LIN {X 0,Y 247.82,Z 1220.634,A -85,B 0,C 180,E1 25956.529,E2 25956.529} C_VEL
LIN {X 0,Y 211.534,Z 1249.474,A -85,B 0,C 180,E1 25974.763,E2 25974.763} C_VEL
LIN {X 0,Y 196.821,Z 1262.562,A -85,B 0,C 180,E1 25994.337,E2 25994.337} C_VEL
LIN {X 0,Y 195.288,Z 1265.442,A -85,B 0,C 180,E1 26012.226,E2 26012.226} C_VEL
LIN {X 0,Y 199.92,Z 1259.369,A -85,B 0,C 180,E1 26032.313,E2 26032.313} C_VEL
LIN {X 0,Y 222.937,Z 1240.033,A -85,B 0,C 180,E1 26052.917,E2 26052.917} C_VEL
LIN {X 0,Y 264.688,Z 1206.28,A -85,B 0,C 180,E1 26068.603,E2 26068.603} C_VEL
LIN {X 0,Y 314.502,Z 1158.82,A -85,B 0,C 180,E1 26078.95,E2 26078.95} C_VEL
LIN {X 0,Y 361.028,Z 1101.859,A -85,B 0,C 180,E1 26085.304,E2 26085.304} C_VEL
LIN {X 0,Y 364.505,Z 1096.146,A -85,B 0,C 180,E1 26086.175,E2 26086.175} C_VEL
LIN {X 0,Y 366.989,Z 1082.941,A -85,B 0,C 180,E1 26094.136,E2 26094.136} C_VEL
LIN {X 0,Y 368.189,Z 1080.031,A -85,B 0,C 180,E1 26101.248,E2 26101.248} C_VEL
LIN {X 0,Y 367.729,Z 1090.519,A -85,B 0,C 180,E1 26110.168,E2 26110.168} C_VEL
LIN {X 0,Y 366.404,Z 1098.087,A -85,B 0,C 180,E1 26113.18,E2 26113.18} C_VEL
LIN {X 0,Y 318.911,Z 1159.271,A -85,B 0,C 180,E1 26119.202,E2 26119.202} C_VEL
LIN {X 0,Y 268.992,Z 1209.566,A -85,B 0,C 180,E1 26128.983,E2 26128.983} C_VEL
LIN {X 0,Y 226.358,Z 1246.346,A -85,B 0,C 180,E1 26143.867,E2 26143.867} C_VEL
LIN {X 0,Y 201.739,Z 1268.464,A -85,B 0,C 180,E1 26163.161,E2 26163.161} C_VEL
LIN {X 0,Y 195.076,Z 1277.751,A -85,B 0,C 180,E1 26183.298,E2 26183.298} C_VEL
LIN {X 0,Y 195.027,Z 1277.758,A -85,B 0,C 180,E1 26196.707,E2 26196.707} C_VEL
LIN {X 0,Y 200.195,Z 1270.124,A -85,B 0,C 180,E1 26214.652,E2 26214.652} C_VEL
LIN {X 0,Y 224.432,Z 1247.98,A -85,B 0,C 180,E1 26235.257,E2 26235.257} C_VEL
LIN {X 0,Y 267.615,Z 1210.892,A -85,B 0,C 180,E1 26250.716,E2 26250.716} C_VEL
LIN {X 0,Y 318.076,Z 1160.468,A -85,B 0,C 180,E1 26260.642,E2 26260.642} C_VEL
LIN {X 0,Y 365.292,Z 1100.027,A -85,B 0,C 180,E1 26266.725,E2 26266.725} C_VEL
LIN {X 0,Y 367.584,Z 1095.292,A -85,B 0,C 180,E1 26267.566,E2 26267.566} C_VEL
LIN {X 0,Y 368.085,Z 1083.099,A -85,B 0,C 180,E1 26275.203,E2 26275.203} C_VEL
LIN {X 0,Y 368.206,Z 1079.906,A -85,B 0,C 180,E1 26281.113,E2 26281.113} C_VEL
LIN {X 0,Y 365.81,Z 1089.05,A -85,B 0,C 180,E1 26290.07,E2 26290.07} C_VEL
LIN {X 0,Y 364.059,Z 1097.903,A -85,B 0,C 180,E1 26294.235,E2 26294.235} C_VEL
LIN {X 0,Y 316.416,Z 1157.039,A -85,B 0,C 180,E1 26300.676,E2 26300.676} C_VEL
LIN {X 0,Y 267.993,Z 1203.645,A -85,B 0,C 180,E1 26310.453,E2 26310.453} C_VEL
LIN {X 0,Y 247.82,Z 1220.634,A -85,B 0,C 180,E1 26316.529,E2 26316.529} C_VEL
LIN {X 0,Y 224.197,Z 1234.966,A -85,B 0,C 180,E1 26321.962,E2 26321.962} C_VEL
LIN {X 0,Y 195.817,Z 1256.691,A -85,B 0,C 180,E1 26341.874,E2 26341.874} C_VEL
LIN {X 0,Y 187.278,Z 1265.309,A -85,B 0,C 180,E1 26363.015,E2 26363.015} C_VEL
LIN {X 0,Y 187.314,Z 1265.279,A -85,B 0,C 180,E1 26376.981,E2 26376.981} C_VEL
LIN {X 0,Y 195.871,Z 1256.598,A -85,B 0,C 180,E1 26398.128,E2 26398.128} C_VEL
LIN {X 0,Y 226.431,Z 1233.395,A -85,B 0,C 180,E1 26418.751,E2 26418.751} C_VEL
LIN {X 0,Y 272.513,Z 1196.349,A -85,B 0,C 180,E1 26433.039,E2 26433.039} C_VEL
LIN {X 0,Y 322.853,Z 1146.97,A -85,B 0,C 180,E1 26442.044,E2 26442.044} C_VEL
LIN {X 0,Y 359.4,Z 1101.578,A -85,B 0,C 180,E1 26446.646,E2 26446.646} C_VEL
LIN {X 0,Y 362.111,Z 1089.495,A -85,B 0,C 180,E1 26454.057,E2 26454.057} C_VEL
LIN {X 0,Y 363.545,Z 1086.616,A -85,B 0,C 180,E1 26461.264,E2 26461.264} C_VEL
LIN {X 0,Y 362.693,Z 1097.481,A -85,B 0,C 180,E1 26470.384,E2 26470.384} C_VEL
LIN {X 0,Y 361.222,Z 1102.92,A -85,B 0,C 180,E1 26472.285,E2 26472.285} C_VEL
LIN {X 0,Y 311.998,Z 1163.707,A -85,B 0,C 180,E1 26478.411,E2 26478.411} C_VEL
LIN {X 0,Y 260.983,Z 1212.827,A -85,B 0,C 180,E1 26488.383,E2 26488.383} C_VEL
LIN {X 0,Y 216.361,Z 1249.506,A -85,B 0,C 180,E1 26504.481,E2 26504.481} C_VEL
LIN {X 0,Y 191.903,Z 1270.717,A -85,B 0,C 180,E1 26525.708,E2 26525.708} C_VEL
LIN {X 0,Y 187.07,Z 1277.486,A -85,B 0,C 180,E1 26543.01,E2 26543.01} C_VEL
LIN {X 0,Y 187.026,Z 1277.494,A -85,B 0,C 180,E1 26556.995,E2 26556.995} C_VEL
LIN {X 0,Y 192.685,Z 1269.852,A -85,B 0,C 180,E1 26575.681,E2 26575.681} C_VEL
LIN {X 0,Y 218.587,Z 1247.704,A -85,B 0,C 180,E1 26596.824,E2 26596.824} C_VEL
LIN {X 0,Y 263.616,Z 1210.619,A -85,B 0,C 180,E1 26612.305,E2 26612.305} C_VEL
LIN {X 0,Y 315.195,Z 1160.441,A -85,B 0,C 180,E1 26622.038,E2 26622.038} C_VEL
LIN {X 0,Y 362.594,Z 1100.59,A -85,B 0,C 180,E1 26628.16,E2 26628.16} C_VEL
LIN {X 0,Y 363.313,Z 1088.664,A -85,B 0,C 180,E1 26636.34,E2 26636.34} C_VEL
LIN {X 0,Y 363.54,Z 1086.485,A -85,B 0,C 180,E1 26641.127,E2 26641.127} C_VEL
LIN {X 0,Y 360.795,Z 1095.869,A -85,B 0,C 180,E1 26650.224,E2 26650.224} C_VEL
LIN {X 0,Y 358.316,Z 1103.36,A -85,B 0,C 180,E1 26653.395,E2 26653.395} C_VEL
LIN {X 0,Y 310.157,Z 1160.831,A -85,B 0,C 180,E1 26659.809,E2 26659.809} C_VEL
LIN {X 0,Y 259.129,Z 1207.77,A -85,B 0,C 180,E1 26670.113,E2 26670.113} C_VEL
LIN {X 0,Y 224.197,Z 1234.966,A -85,B 0,C 180,E1 26681.962,E2 26681.962} C_VEL
LIN {X 0,Y 202.634,Z 1246.721,A -85,B 0,C 180,E1 26688.863,E2 26688.863} C_VEL
LIN {X 0,Y 183.451,Z 1261.13,A -85,B 0,C 180,E1 26708.135,E2 26708.135} C_VEL
LIN {X 0,Y 179.089,Z 1265.984,A -85,B 0,C 180,E1 26727.569,E2 26727.569} C_VEL
LIN {X 0,Y 181.319,Z 1263.044,A -85,B 0,C 180,E1 26747.039,E2 26747.039} C_VEL
LIN {X 0,Y 200.823,Z 1247.851,A -85,B 0,C 180,E1 26769.981,E2 26769.981} C_VEL
LIN {X 0,Y 242.467,Z 1217.738,A -85,B 0,C 180,E1 26787.99,E2 26787.99} C_VEL
LIN {X 0,Y 294.507,Z 1173.617,A -85,B 0,C 180,E1 26799.507,E2 26799.507} C_VEL
LIN {X 0,Y 345.516,Z 1117.781,A -85,B 0,C 180,E1 26806.587,E2 26806.587} C_VEL
LIN {X 0,Y 354.577,Z 1105.763,A -85,B 0,C 180,E1 26807.709,E2 26807.709} C_VEL
LIN {X 0,Y 357.614,Z 1094.475,A -85,B 0,C 180,E1 26816.024,E2 26816.024} C_VEL
LIN {X 0,Y 358.71,Z 1093.075,A -85,B 0,C 180,E1 26821.281,E2 26821.281} C_VEL
LIN {X 0,Y 357.6,Z 1104.102,A -85,B 0,C 180,E1 26830.46,E2 26830.46} C_VEL
LIN {X 0,Y 354.697,Z 1109.234,A -85,B 0,C 180,E1 26831.485,E2 26831.485} C_VEL
LIN {X 0,Y 304.591,Z 1168.393,A -85,B 0,C 180,E1 26837.656,E2 26837.656} C_VEL
LIN {X 0,Y 252.665,Z 1216.169,A -85,B 0,C 180,E1 26847.835,E2 26847.835} C_VEL
LIN {X 0,Y 207.148,Z 1251.806,A -85,B 0,C 180,E1 26864.675,E2 26864.675} C_VEL
LIN {X 0,Y 184.346,Z 1270.499,A -85,B 0,C 180,E1 26884.752,E2 26884.752} C_VEL
LIN {X 0,Y 179.063,Z 1277.221,A -85,B 0,C 180,E1 26902.695,E2 26902.695} C_VEL
LIN {X 0,Y 179.022,Z 1277.229,A -85,B 0,C 180,E1 26917.309,E2 26917.309} C_VEL
LIN {X 0,Y 185.224,Z 1269.58,A -85,B 0,C 180,E1 26936.796,E2 26936.796} C_VEL
LIN {X 0,Y 212.914,Z 1247.429,A -85,B 0,C 180,E1 26958.477,E2 26958.477} C_VEL
LIN {X 0,Y 259.603,Z 1210.534,A -85,B 0,C 180,E1 26973.896,E2 26973.896} C_VEL
LIN {X 0,Y 312.717,Z 1160.17,A -85,B 0,C 180,E1 26983.496,E2 26983.496} C_VEL
LIN {X 0,Y 357.527,Z 1105.477,A -85,B 0,C 180,E1 26988.92,E2 26988.92} C_VEL
LIN {X 0,Y 358.49,Z 1095.118,A -85,B 0,C 180,E1 26996.29,E2 26996.29} C_VEL
LIN {X 0,Y 358.707,Z 1092.939,A -85,B 0,C 180,E1 27001.142,E2 27001.142} C_VEL
LIN {X 0,Y 355.546,Z 1102.56,A -85,B 0,C 180,E1 27010.377,E2 27010.377} C_VEL
LIN {X 0,Y 354.073,Z 1106.906,A -85,B 0,C 180,E1 27012.377,E2 27012.377} C_VEL
LIN {X 0,Y 304.521,Z 1164.053,A -85,B 0,C 180,E1 27018.809,E2 27018.809} C_VEL
LIN {X 0,Y 252.236,Z 1210.301,A -85,B 0,C 180,E1 27029.224,E2 27029.224} C_VEL
LIN {X 0,Y 207.365,Z 1243.323,A -85,B 0,C 180,E1 27045.932,E2 27045.932} C_VEL
LIN {X 0,Y 202.634,Z 1246.721,A -85,B 0,C 180,E1 27048.863,E2 27048.863} C_VEL
LIN {X 0,Y 183.392,Z 1255.903,A -85,B 0,C 180,E1 27057.335,E2 27057.335} C_VEL
LIN {X 0,Y 171.965,Z 1264.872,A -85,B 0,C 180,E1 27077.248,E2 27077.248} C_VEL
LIN {X 0,Y 171.252,Z 1266.232,A -85,B 0,C 180,E1 27092.539,E2 27092.539} C_VEL
LIN {X 0,Y 177.324,Z 1260.268,A -85,B 0,C 180,E1 27115.128,E2 27115.128} C_VEL
LIN {X 0,Y 205.419,Z 1240.853,A -85,B 0,C 180,E1 27137.647,E2 27137.647} C_VEL
LIN {X 0,Y 253.016,Z 1206.793,A -85,B 0,C 180,E1 27153.526,E2 27153.526} C_VEL
LIN {X 0,Y 307.106,Z 1159.027,A -85,B 0,C 180,E1 27163.364,E2 27163.364} C_VEL
LIN {X 0,Y 349.8,Z 1110.023,A -85,B 0,C 180,E1 27168.818,E2 27168.818} C_VEL
LIN {X 0,Y 352.834,Z 1100.625,A -85,B 0,C 180,E1 27176.373,E2 27176.373} C_VEL
LIN {X 0,Y 353.886,Z 1099.52,A -85,B 0,C 180,E1 27181.299,E2 27181.299} C_VEL
LIN {X 0,Y 352.404,Z 1109.662,A -85,B 0,C 180,E1 27190.053,E2 27190.053} C_VEL
LIN {X 0,Y 300.349,Z 1169.933,A -85,B 0,C 180,E1 27196.404,E2 27196.404} C_VEL
LIN {X 0,Y 246.438,Z 1217.829,A -85,B 0,C 180,E1 27206.72,E2 27206.72} C_VEL
LIN {X 0,Y 199.799,Z 1252.653,A -85,B 0,C 180,E1 27223.796,E2 27223.796} C_VEL
LIN {X 0,Y 174.925,Z 1271.959,A -85,B 0,C 180,E1 27247.013,E2 27247.013} C_VEL
LIN {X 0,Y 171.215,Z 1277.464,A -85,B 0,C 180,E1 27267.461,E2 27267.461} C_VEL
LIN {X 0,Y 171.634,Z 1275.862,A -85,B 0,C 180,E1 27282.777,E2 27282.777} C_VEL
LIN {X 0,Y 184.77,Z 1263.609,A -85,B 0,C 180,E1 27305.855,E2 27305.855} C_VEL
LIN {X 0,Y 223.269,Z 1235.666,A -85,B 0,C 180,E1 27326.404,E2 27326.404} C_VEL
LIN {X 0,Y 275.503,Z 1193.538,A -85,B 0,C 180,E1 27339.512,E2 27339.512} C_VEL
LIN {X 0,Y 328.814,Z 1139.598,A -85,B 0,C 180,E1 27347.25,E2 27347.25} C_VEL
LIN {X 0,Y 352.52,Z 1109.78,A -85,B 0,C 180,E1 27349.969,E2 27349.969} C_VEL
LIN {X 0,Y 353.968,Z 1099.785,A -85,B 0,C 180,E1 27358.701,E2 27358.701} C_VEL
LIN {X 0,Y 352.024,Z 1103.065,A -85,B 0,C 180,E1 27366.114,E2 27366.114} C_VEL
LIN {X 0,Y 348.563,Z 1112.301,A -85,B 0,C 180,E1 27371.487,E2 27371.487} C_VEL
LIN {X 0,Y 296.977,Z 1169.258,A -85,B 0,C 180,E1 27378.071,E2 27378.071} C_VEL
LIN {X 0,Y 244.238,Z 1213.752,A -85,B 0,C 180,E1 27388.599,E2 27388.599} C_VEL
LIN {X 0,Y 198.822,Z 1245.441,A -85,B 0,C 180,E1 27405.798,E2 27405.798} C_VEL
LIN {X 0,Y 183.392,Z 1255.903,A -85,B 0,C 180,E1 27417.335,E2 27417.335} C_VEL
LIN {X 0,Y 167.503,Z 1262.23,A -85,B 0,C 180,E1 27427.557,E2 27427.557} C_VEL
LIN {X 0,Y 163.087,Z 1266.509,A -85,B 0,C 180,E1 27447.331,E2 27447.331} C_VEL
LIN {X 0,Y 164.522,Z 1264.699,A -85,B 0,C 180,E1 27465.063,E2 27465.063} C_VEL
LIN {X 0,Y 182.018,Z 1252.531,A -85,B 0,C 180,E1 27488.72,E2 27488.72} C_VEL
LIN {X 0,Y 223.224,Z 1225.893,A -85,B 0,C 180,E1 27508.221,E2 27508.221} C_VEL
LIN {X 0,Y 275.947,Z 1185.814,A -85,B 0,C 180,E1 27520.409,E2 27520.409} C_VEL
LIN {X 0,Y 329.244,Z 1133.47,A -85,B 0,C 180,E1 27527.862,E2 27527.862} C_VEL
LIN {X 0,Y 345.057,Z 1114.374,A -85,B 0,C 180,E1 27529.945,E2 27529.945} C_VEL
LIN {X 0,Y 348.705,Z 1105.384,A -85,B 0,C 180,E1 27538.845,E2 27538.845} C_VEL
LIN {X 0,Y 347.695,Z 1111.993,A -85,B 0,C 180,E1 27547.587,E2 27547.587} C_VEL
LIN {X 0,Y 346.201,Z 1116.091,A -85,B 0,C 180,E1 27549.381,E2 27549.381} C_VEL
LIN {X 0,Y 293.651,Z 1174.078,A -85,B 0,C 180,E1 27555.5,E2 27555.5} C_VEL
LIN {X 0,Y 239.428,Z 1220.197,A -85,B 0,C 180,E1 27565.775,E2 27565.775} C_VEL
LIN {X 0,Y 192.133,Z 1253.758,A -85,B 0,C 180,E1 27583.042,E2 27583.042} C_VEL
LIN {X 0,Y 167.404,Z 1271.689,A -85,B 0,C 180,E1 27605.917,E2 27605.917} C_VEL
LIN {X 0,Y 163.19,Z 1277.2,A -85,B 0,C 180,E1 27627.336,E2 27627.336} C_VEL
LIN {X 0,Y 163.731,Z 1275.596,A -85,B 0,C 180,E1 27643.405,E2 27643.405} C_VEL
LIN {X 0,Y 178.813,Z 1262.852,A -85,B 0,C 180,E1 27667.992,E2 27667.992} C_VEL
LIN {X 0,Y 220.389,Z 1234.213,A -85,B 0,C 180,E1 27688.783,E2 27688.783} C_VEL
LIN {X 0,Y 274.235,Z 1191.905,A -85,B 0,C 180,E1 27701.446,E2 27701.446} C_VEL
LIN {X 0,Y 328.798,Z 1137.381,A -85,B 0,C 180,E1 27708.862,E2 27708.862} C_VEL
LIN {X 0,Y 347.578,Z 1114.028,A -85,B 0,C 180,E1 27711.139,E2 27711.139} C_VEL
LIN {X 0,Y 348.89,Z 1106.026,A -85,B 0,C 180,E1 27718.683,E2 27718.683} C_VEL
LIN {X 0,Y 346.809,Z 1109.446,A -85,B 0,C 180,E1 27726.206,E2 27726.206} C_VEL
LIN {X 0,Y 343.981,Z 1116.331,A -85,B 0,C 180,E1 27730.466,E2 27730.466} C_VEL
LIN {X 0,Y 291.649,Z 1172.1,A -85,B 0,C 180,E1 27736.964,E2 27736.964} C_VEL
LIN {X 0,Y 238.969,Z 1214.983,A -85,B 0,C 180,E1 27747.201,E2 27747.201} C_VEL
LIN {X 0,Y 193.421,Z 1245.414,A -85,B 0,C 180,E1 27763.783,E2 27763.783} C_VEL
LIN {X 0,Y 167.503,Z 1262.23,A -85,B 0,C 180,E1 27787.557,E2 27787.557} C_VEL
LIN {X 0,Y 155.495,Z 1265.989,A -85,B 0,C 180,E1 27799.357,E2 27799.357} C_VEL
LIN {X 0,Y 155.363,Z 1266.338,A -85,B 0,C 180,E1 27818.427,E2 27818.427} C_VEL
LIN {X 0,Y 167.147,Z 1257.93,A -85,B 0,C 180,E1 27843.019,E2 27843.019} C_VEL
LIN {X 0,Y 206.316,Z 1234.282,A -85,B 0,C 180,E1 27865.871,E2 27865.871} C_VEL
LIN {X 0,Y 260.188,Z 1196.663,A -85,B 0,C 180,E1 27879.779,E2 27879.779} C_VEL
LIN {X 0,Y 315.943,Z 1146.366,A -85,B 0,C 180,E1 27887.952,E2 27887.952} C_VEL
LIN {X 0,Y 339.961,Z 1119.245,A -85,B 0,C 180,E1 27890.746,E2 27890.746} C_VEL
LIN {X 0,Y 343.594,Z 1111.606,A -85,B 0,C 180,E1 27898.832,E2 27898.832} C_VEL
LIN {X 0,Y 342.731,Z 1116.701,A -85,B 0,C 180,E1 27906.427,E2 27906.427} C_VEL
LIN {X 0,Y 340.761,Z 1120.982,A -85,B 0,C 180,E1 27908.405,E2 27908.405} C_VEL
LIN {X 0,Y 286.348,Z 1178.518,A -85,B 0,C 180,E1 27914.64,E2 27914.64} C_VEL
LIN {X 0,Y 231.031,Z 1223.386,A -85,B 0,C 180,E1 27925.127,E2 27925.127} C_VEL
LIN {X 0,Y 182.577,Z 1255.896,A -85,B 0,C 180,E1 27943.32,E2 27943.32} C_VEL
LIN {X 0,Y 158.534,Z 1272.684,A -85,B 0,C 180,E1 27967.48,E2 27967.48} C_VEL
LIN {X 0,Y 155.186,Z 1276.937,A -85,B 0,C 180,E1 27987.198,E2 27987.198} C_VEL
LIN {X 0,Y 155.82,Z 1275.329,A -85,B 0,C 180,E1 28004.099,E2 28004.099} C_VEL
LIN {X 0,Y 172.329,Z 1262.579,A -85,B 0,C 180,E1 28029.696,E2 28029.696} C_VEL
LIN {X 0,Y 215.441,Z 1234.41,A -85,B 0,C 180,E1 28050.479,E2 28050.479} C_VEL
LIN {X 0,Y 271.676,Z 1191.631,A -85,B 0,C 180,E1 28063.128,E2 28063.128} C_VEL
LIN {X 0,Y 327.296,Z 1137.112,A -85,B 0,C 180,E1 28070.287,E2 28070.287} C_VEL
LIN {X 0,Y 342.517,Z 1118.724,A -85,B 0,C 180,E1 28072.134,E2 28072.134} C_VEL
LIN {X 0,Y 343.762,Z 1112.266,A -85,B 0,C 180,E1 28078.663,E2 28078.663} C_VEL
LIN {X 0,Y 342.129,Z 1114.45,A -85,B 0,C 180,E1 28084.888,E2 28084.888} C_VEL
LIN {X 0,Y 339.03,Z 1120.817,A -85,B 0,C 180,E1 28089.466,E2 28089.466} C_VEL
LIN {X 0,Y 284.444,Z 1176.685,A -85,B 0,C 180,E1 28096.116,E2 28096.116} C_VEL
LIN {X 0,Y 229.669,Z 1219.072,A -85,B 0,C 180,E1 28106.827,E2 28106.827} C_VEL
LIN {X 0,Y 182.459,Z 1248.784,A -85,B 0,C 180,E1 28124.988,E2 28124.988} C_VEL
LIN {X 0,Y 158.066,Z 1263.894,A -85,B 0,C 180,E1 28150.356,E2 28150.356} C_VEL
LIN {X 0,Y 155.495,Z 1265.989,A -85,B 0,C 180,E1 28159.357,E2 28159.357} C_VEL
LIN {X 0,Y 147.144,Z 1267.023,A -85,B 0,C 180,E1 28172.526,E2 28172.526} C_VEL
LIN {X 0,Y 153.59,Z 1262.14,A -85,B 0,C 180,E1 28196.408,E2 28196.408} C_VEL
LIN {X 0,Y 185,Z 1244.276,A -85,B 0,C 180,E1 28221.219,E2 28221.219} C_VEL
LIN {X 0,Y 236.27,Z 1212.304,A -85,B 0,C 180,E1 28237.409,E2 28237.409} C_VEL
LIN {X 0,Y 294.045,Z 1166.277,A -85,B 0,C 180,E1 28247.02,E2 28247.02} C_VEL
LIN {X 0,Y 335.073,Z 1123.776,A -85,B 0,C 180,E1 28251.822,E2 28251.822} C_VEL
LIN {X 0,Y 338.374,Z 1117.761,A -85,B 0,C 180,E1 28258.819,E2 28258.819} C_VEL
LIN {X 0,Y 337.028,Z 1123.748,A -85,B 0,C 180,E1 28267.186,E2 28267.186} C_VEL
LIN {X 0,Y 280.986,Z 1181.213,A -85,B 0,C 180,E1 28273.47,E2 28273.47} C_VEL
LIN {X 0,Y 222.866,Z 1226.333,A -85,B 0,C 180,E1 28284.348,E2 28284.348} C_VEL
LIN {X 0,Y 174.905,Z 1256.809,A -85,B 0,C 180,E1 28302.46,E2 28302.46} C_VEL
LIN {X 0,Y 149.72,Z 1273.343,A -85,B 0,C 180,E1 28329.215,E2 28329.215} C_VEL
LIN {X 0,Y 147.157,Z 1276.673,A -85,B 0,C 180,E1 28347.045,E2 28347.045} C_VEL
LIN {X 0,Y 147.952,Z 1275.062,A -85,B 0,C 180,E1 28364.866,E2 28364.866} C_VEL
LIN {X 0,Y 165.982,Z 1262.306,A -85,B 0,C 180,E1 28391.539,E2 28391.539} C_VEL
LIN {X 0,Y 210.575,Z 1234.685,A -85,B 0,C 180,E1 28412.22,E2 28412.22} C_VEL
LIN {X 0,Y 267.272,Z 1193.074,A -85,B 0,C 180,E1 28424.517,E2 28424.517} C_VEL
LIN {X 0,Y 323.749,Z 1139.311,A -85,B 0,C 180,E1 28431.507,E2 28431.507} C_VEL
LIN {X 0,Y 337.26,Z 1123.525,A -85,B 0,C 180,E1 28433.061,E2 28433.061} C_VEL
LIN {X 0,Y 338.437,Z 1118.009,A -85,B 0,C 180,E1 28441.211,E2 28441.211} C_VEL
LIN {X 0,Y 334.075,Z 1125.433,A -85,B 0,C 180,E1 28448.451,E2 28448.451} C_VEL
LIN {X 0,Y 278.957,Z 1179.832,A -85,B 0,C 180,E1 28454.985,E2 28454.985} C_VEL
LIN {X 0,Y 222.567,Z 1221.67,A -85,B 0,C 180,E1 28465.832,E2 28465.832} C_VEL
LIN {X 0,Y 174.764,Z 1250.167,A -85,B 0,C 180,E1 28484.219,E2 28484.219} C_VEL
LIN {X 0,Y 150.414,Z 1264.161,A -85,B 0,C 180,E1 28509.312,E2 28509.312} C_VEL
LIN {X 0,Y 147.144,Z 1267.023,A -85,B 0,C 180,E1 28532.526,E2 28532.526} C_VEL
LIN {X 0,Y 140.79,Z 1265.707,A -85,B 0,C 180,E1 28546.477,E2 28546.477} C_VEL
LIN {X 0,Y 163.307,Z 1253.352,A -85,B 0,C 180,E1 28574.201,E2 28574.201} C_VEL
LIN {X 0,Y 211.07,Z 1226.722,A -85,B 0,C 180,E1 28594.032,E2 28594.032} C_VEL
LIN {X 0,Y 268.221,Z 1186.962,A -85,B 0,C 180,E1 28605.35,E2 28605.35} C_VEL
LIN {X 0,Y 325.224,Z 1134.001,A -85,B 0,C 180,E1 28612.143,E2 28612.143} C_VEL
LIN {X 0,Y 330.195,Z 1128.455,A -85,B 0,C 180,E1 28612.888,E2 28612.888} C_VEL
LIN {X 0,Y 332.972,Z 1123.76,A -85,B 0,C 180,E1 28618.804,E2 28618.804} C_VEL
LIN {X 0,Y 331.949,Z 1128.073,A -85,B 0,C 180,E1 28625.829,E2 28625.829} C_VEL
LIN {X 0,Y 275.731,Z 1183.905,A -85,B 0,C 180,E1 28632.242,E2 28632.242} C_VEL
LIN {X 0,Y 216.253,Z 1228.257,A -85,B 0,C 180,E1 28643.136,E2 28643.136} C_VEL
LIN {X 0,Y 165.269,Z 1258.916,A -85,B 0,C 180,E1 28662.711,E2 28662.711} C_VEL
LIN {X 0,Y 142.073,Z 1273.073,A -85,B 0,C 180,E1 28688.04,E2 28688.04} C_VEL
LIN {X 0,Y 139.141,Z 1276.41,A -85,B 0,C 180,E1 28706.875,E2 28706.875} C_VEL
LIN {X 0,Y 140.085,Z 1274.795,A -85,B 0,C 180,E1 28725.721,E2 28725.721} C_VEL
LIN {X 0,Y 159.805,Z 1262.031,A -85,B 0,C 180,E1 28753.532,E2 28753.532} C_VEL
LIN {X 0,Y 207.096,Z 1234.18,A -85,B 0,C 180,E1 28774.412,E2 28774.412} C_VEL
LIN {X 0,Y 266.581,Z 1191.655,A -85,B 0,C 180,E1 28786.47,E2 28786.47} C_VEL
LIN {X 0,Y 324.204,Z 1137.327,A -85,B 0,C 180,E1 28793.118,E2 28793.118} C_VEL
LIN {X 0,Y 332.123,Z 1128.152,A -85,B 0,C 180,E1 28794.184,E2 28794.184} C_VEL
LIN {X 0,Y 333.023,Z 1124.019,A -85,B 0,C 180,E1 28801.23,E2 28801.23} C_VEL
LIN {X 0,Y 329.154,Z 1130.096,A -85,B 0,C 180,E1 28807.418,E2 28807.418} C_VEL
LIN {X 0,Y 273.568,Z 1182.952,A -85,B 0,C 180,E1 28813.796,E2 28813.796} C_VEL
LIN {X 0,Y 216.416,Z 1223.676,A -85,B 0,C 180,E1 28824.534,E2 28824.534} C_VEL
LIN {X 0,Y 166.296,Z 1251.987,A -85,B 0,C 180,E1 28843.903,E2 28843.903} C_VEL
LIN {X 0,Y 142.812,Z 1264.429,A -85,B 0,C 180,E1 28868.156,E2 28868.156} C_VEL
LIN {X 0,Y 139.149,Z 1267.286,A -85,B 0,C 180,E1 28892.699,E2 28892.699} C_VEL
LIN {X 0,Y 140.79,Z 1265.707,A -85,B 0,C 180,E1 28906.477,E2 28906.477} C_VEL
LIN {X 0,Y 140.196,Z 1262.119,A -85,B 0,C 180,E1 28920.901,E2 28920.901} C_VEL
LIN {X 0,Y 177.465,Z 1243.583,A -85,B 0,C 180,E1 28946.41,E2 28946.41} C_VEL
LIN {X 0,Y 235.248,Z 1209.608,A -85,B 0,C 180,E1 28962.145,E2 28962.145} C_VEL
LIN {X 0,Y 294.291,Z 1163.658,A -85,B 0,C 180,E1 28970.595,E2 28970.595} C_VEL
LIN {X 0,Y 325.081,Z 1133.303,A -85,B 0,C 180,E1 28973.769,E2 28973.769} C_VEL
LIN {X 0,Y 327.566,Z 1129.763,A -85,B 0,C 180,E1 28978.789,E2 28978.789} C_VEL
LIN {X 0,Y 325.946,Z 1133.997,A -85,B 0,C 180,E1 28985.206,E2 28985.206} C_VEL
LIN {X 0,Y 267.563,Z 1188.977,A -85,B 0,C 180,E1 28991.362,E2 28991.362} C_VEL
LIN {X 0,Y 208.025,Z 1231.096,A -85,B 0,C 180,E1 29002.246,E2 29002.246} C_VEL
LIN {X 0,Y 155.63,Z 1260.699,A -85,B 0,C 180,E1 29022.982,E2 29022.982} C_VEL
LIN {X 0,Y 134.486,Z 1272.803,A -85,B 0,C 180,E1 29046.73,E2 29046.73} C_VEL
LIN {X 0,Y 131.109,Z 1276.146,A -85,B 0,C 180,E1 29066.683,E2 29066.683} C_VEL
LIN {X 0,Y 132.273,Z 1274.528,A -85,B 0,C 180,E1 29086.676,E2 29086.676} C_VEL
LIN {X 0,Y 155.758,Z 1260.753,A -85,B 0,C 180,E1 29116.973,E2 29116.973} C_VEL
LIN {X 0,Y 205.878,Z 1232.497,A -85,B 0,C 180,E1 29137.184,E2 29137.184} C_VEL
LIN {X 0,Y 265.764,Z 1190.573,A -85,B 0,C 180,E1 29148.378,E2 29148.378} C_VEL
LIN {X 0,Y 324.358,Z 1135.947,A -85,B 0,C 180,E1 29154.664,E2 29154.664} C_VEL
LIN {X 0,Y 327.157,Z 1132.196,A -85,B 0,C 180,E1 29156.1,E2 29156.1} C_VEL
LIN {X 0,Y 326.784,Z 1130.961,A -85,B 0,C 180,E1 29162.778,E2 29162.778} C_VEL
LIN {X 0,Y 324.208,Z 1134.549,A -85,B 0,C 180,E1 29166.349,E2 29166.349} C_VEL
LIN {X 0,Y 266.672,Z 1187.08,A -85,B 0,C 180,E1 29172.769,E2 29172.769} C_VEL
LIN {X 0,Y 207.521,Z 1227.149,A -85,B 0,C 180,E1 29183.871,E2 29183.871} C_VEL
LIN {X 0,Y 157.492,Z 1253.714,A -85,B 0,C 180,E1 29203.699,E2 29203.699} C_VEL
LIN {X 0,Y 132.756,Z 1266.2,A -85,B 0,C 180,E1 29233.386,E2 29233.386} C_VEL
LIN {X 0,Y 131.192,Z 1267.548,A -85,B 0,C 180,E1 29253.315,E2 29253.315} C_VEL
LIN {X 0,Y 140.196,Z 1262.119,A -85,B 0,C 180,E1 29280.901,E2 29280.901} C_VEL
LIN {X 0,Y 146.198,Z 1256.511,A -85,B 0,C 180,E1 29294.795,E2 29294.795} C_VEL
LIN {X 0,Y 195.43,Z 1232.359,A -85,B 0,C 180,E1 29315.885,E2 29315.885} C_VEL
LIN {X 0,Y 256.36,Z 1193.718,A -85,B 0,C 180,E1 29327.71,E2 29327.71} C_VEL
LIN {X 0,Y 315.759,Z 1142.496,A -85,B 0,C 180,E1 29334.358,E2 29334.358} C_VEL
LIN {X 0,Y 320.078,Z 1137.873,A -85,B 0,C 180,E1 29335.115,E2 29335.115} C_VEL
LIN {X 0,Y 322.048,Z 1135.97,A -85,B 0,C 180,E1 29341.427,E2 29341.427} C_VEL
LIN {X 0,Y 318.728,Z 1140.662,A -85,B 0,C 180,E1 29344.284,E2 29344.284} C_VEL
LIN {X 0,Y 259.057,Z 1194.108,A -85,B 0,C 180,E1 29350.484,E2 29350.484} C_VEL
LIN {X 0,Y 196.629,Z 1235.696,A -85,B 0,C 180,E1 29362.11,E2 29362.11} C_VEL
LIN {X 0,Y 144.94,Z 1262.985,A -85,B 0,C 180,E1 29384.048,E2 29384.048} C_VEL
LIN {X 0,Y 124.468,Z 1274.247,A -85,B 0,C 180,E1 29412.249,E2 29412.249} C_VEL
LIN {X 0,Y 122.974,Z 1275.882,A -85,B 0,C 180,E1 29433.541,E2 29433.541} C_VEL
LIN {X 0,Y 130.735,Z 1270.36,A -85,B 0,C 180,E1 29461.506,E2 29461.506} C_VEL
LIN {X 0,Y 168.66,Z 1251.051,A -85,B 0,C 180,E1 29488.774,E2 29488.774} C_VEL
LIN {X 0,Y 228.181,Z 1216.274,A -85,B 0,C 180,E1 29504.736,E2 29504.736} C_VEL
LIN {X 0,Y 290.528,Z 1168.213,A -85,B 0,C 180,E1 29513.137,E2 29513.137} C_VEL
LIN {X 0,Y 320.168,Z 1139.396,A -85,B 0,C 180,E1 29515.846,E2 29515.846} C_VEL
LIN {X 0,Y 321.96,Z 1135.823,A -85,B 0,C 180,E1 29521.273,E2 29521.273} C_VEL
LIN {X 0,Y 318.829,Z 1139.572,A -85,B 0,C 180,E1 29525.293,E2 29525.293} C_VEL
LIN {X 0,Y 259.713,Z 1191.318,A -85,B 0,C 180,E1 29531.7,E2 29531.7} C_VEL
LIN {X 0,Y 198.291,Z 1230.818,A -85,B 0,C 180,E1 29543.257,E2 29543.257} C_VEL
LIN {X 0,Y 147.83,Z 1255.842,A -85,B 0,C 180,E1 29564.037,E2 29564.037} C_VEL
LIN {X 0,Y 124.992,Z 1266.467,A -85,B 0,C 180,E1 29592.321,E2 29592.321} C_VEL
LIN {X 0,Y 123.204,Z 1267.811,A -85,B 0,C 180,E1 29613.53,E2 29613.53} C_VEL
LIN {X 0,Y 134.585,Z 1261.797,A -85,B 0,C 180,E1 29644.331,E2 29644.331} C_VEL
LIN {X 0,Y 146.198,Z 1256.511,A -85,B 0,C 180,E1 29654.795,E2 29654.795} C_VEL
LIN {X 0,Y 158.407,Z 1248.902,A -85,B 0,C 180,E1 29667.052,E2 29667.052} C_VEL
LIN {X 0,Y 217.337,Z 1218.399,A -85,B 0,C 180,E1 29683.758,E2 29683.758} C_VEL
LIN {X 0,Y 279.244,Z 1175.075,A -85,B 0,C 180,E1 29692.471,E2 29692.471} C_VEL
LIN {X 0,Y 314.799,Z 1143.012,A -85,B 0,C 180,E1 29695.934,E2 29695.934} C_VEL
LIN {X 0,Y 316.074,Z 1142.36,A -85,B 0,C 180,E1 29702.356,E2 29702.356} C_VEL
LIN {X 0,Y 311.727,Z 1147.09,A -85,B 0,C 180,E1 29703.303,E2 29703.303} C_VEL
LIN {X 0,Y 250.202,Z 1199.406,A -85,B 0,C 180,E1 29709.612,E2 29709.612} C_VEL
LIN {X 0,Y 186.549,Z 1239.293,A -85,B 0,C 180,E1 29721.612,E2 29721.612} C_VEL
LIN {X 0,Y 136.379,Z 1264.072,A -85,B 0,C 180,E1 29743.654,E2 29743.654} C_VEL
LIN {X 0,Y 116.708,Z 1273.979,A -85,B 0,C 180,E1 29771.025,E2 29771.025} C_VEL
LIN {X 0,Y 114.944,Z 1275.618,A -85,B 0,C 180,E1 29793.789,E2 29793.789} C_VEL
LIN {X 0,Y 123.726,Z 1270.088,A -85,B 0,C 180,E1 29823.517,E2 29823.517} C_VEL
LIN {X 0,Y 164.454,Z 1250.776,A -85,B 0,C 180,E1 29851.282,E2 29851.282} C_VEL
LIN {X 0,Y 226.124,Z 1216.001,A -85,B 0,C 180,E1 29866.78,E2 29866.78} C_VEL
LIN {X 0,Y 289.651,Z 1167.942,A -85,B 0,C 180,E1 29874.774,E2 29874.774} C_VEL
LIN {X 0,Y 316.045,Z 1142.855,A -85,B 0,C 180,E1 29877.196,E2 29877.196} C_VEL
LIN {X 0,Y 316.261,Z 1141.601,A -85,B 0,C 180,E1 29881.295,E2 29881.295} C_VEL
LIN {X 0,Y 313.598,Z 1144.555,A -85,B 0,C 180,E1 29884.202,E2 29884.202} C_VEL
LIN {X 0,Y 252.892,Z 1195.476,A -85,B 0,C 180,E1 29890.575,E2 29890.575} C_VEL
LIN {X 0,Y 191.801,Z 1232.946,A -85,B 0,C 180,E1 29901.862,E2 29901.862} C_VEL
LIN {X 0,Y 138.157,Z 1257.863,A -85,B 0,C 180,E1 29924.416,E2 29924.416} C_VEL
LIN {X 0,Y 115.579,Z 1267.689,A -85,B 0,C 180,E1 29958.635,E2 29958.635} C_VEL
LIN {X 0,Y 115.617,Z 1267.663,A -85,B 0,C 180,E1 29981.357,E2 29981.357} C_VEL
LIN {X 0,Y 138.193,Z 1257.791,A -85,B 0,C 180,E1 30015.563,E2 30015.563} C_VEL
LIN {X 0,Y 158.407,Z 1248.902,A -85,B 0,C 180,E1 30027.052,E2 30027.052} C_VEL
LIN {X 0,Y 176.251,Z 1239.257,A -85,B 0,C 180,E1 30037.079,E2 30037.079} C_VEL
LIN {X 0,Y 239.264,Z 1203.822,A -85,B 0,C 180,E1 30049.56,E2 30049.56} C_VEL
LIN {X 0,Y 300.489,Z 1156.372,A -85,B 0,C 180,E1 30056.186,E2 30056.186} C_VEL
LIN {X 0,Y 309.611,Z 1147.81,A -85,B 0,C 180,E1 30057.272,E2 30057.272} C_VEL
LIN {X 0,Y 309.769,Z 1148.324,A -85,B 0,C 180,E1 30061.896,E2 30061.896} C_VEL
LIN {X 0,Y 248.929,Z 1199.126,A -85,B 0,C 180,E1 30067.691,E2 30067.691} C_VEL
LIN {X 0,Y 184.558,Z 1238.538,A -85,B 0,C 180,E1 30078.928,E2 30078.928} C_VEL
LIN {X 0,Y 130.732,Z 1263.796,A -85,B 0,C 180,E1 30100.994,E2 30100.994} C_VEL
LIN {X 0,Y 109.005,Z 1273.71,A -85,B 0,C 180,E1 30129.627,E2 30129.627} C_VEL
LIN {X 0,Y 106.927,Z 1275.355,A -85,B 0,C 180,E1 30154.073,E2 30154.073} C_VEL
LIN {X 0,Y 116.884,Z 1269.815,A -85,B 0,C 180,E1 30185.768,E2 30185.768} C_VEL
LIN {X 0,Y 162.74,Z 1249.464,A -85,B 0,C 180,E1 30214.653,E2 30214.653} C_VEL
LIN {X 0,Y 227.385,Z 1213.76,A -85,B 0,C 180,E1 30229.372,E2 30229.372} C_VEL
LIN {X 0,Y 290.688,Z 1166.198,A -85,B 0,C 180,E1 30236.564,E2 30236.564} C_VEL
LIN {X 0,Y 310.69,Z 1147.589,A -85,B 0,C 180,E1 30238.521,E2 30238.521} C_VEL
LIN {X 0,Y 309.567,Z 1148.119,A -85,B 0,C 180,E1 30242.728,E2 30242.728} C_VEL
LIN {X 0,Y 247.923,Z 1198.144,A -85,B 0,C 180,E1 30249.182,E2 30249.182} C_VEL
LIN {X 0,Y 183.561,Z 1235.764,A -85,B 0,C 180,E1 30260.829,E2 30260.829} C_VEL
LIN {X 0,Y 129.511,Z 1259.216,A -85,B 0,C 180,E1 30283.972,E2 30283.972} C_VEL
LIN {X 0,Y 107.664,Z 1267.954,A -85,B 0,C 180,E1 30317.787,E2 30317.787} C_VEL
LIN {X 0,Y 107.702,Z 1267.929,A -85,B 0,C 180,E1 30342.204,E2 30342.204} C_VEL
LIN {X 0,Y 129.936,Z 1259.02,A -85,B 0,C 180,E1 30376.22,E2 30376.22} C_VEL
LIN {X 0,Y 176.251,Z 1239.257,A -85,B 0,C 180,E1 30397.079,E2 30397.079} C_VEL
LIN {X 0,Y 197.144,Z 1227.732,A -85,B 0,C 180,E1 30405.171,E2 30405.171} C_VEL
LIN {X 0,Y 263.111,Z 1186.702,A -85,B 0,C 180,E1 30414.435,E2 30414.435} C_VEL
LIN {X 0,Y 304.277,Z 1152.737,A -85,B 0,C 180,E1 30418.297,E2 30418.297} C_VEL
LIN {X 0,Y 303.344,Z 1153.944,A -85,B 0,C 180,E1 30420.801,E2 30420.801} C_VEL
LIN {X 0,Y 240.717,Z 1203.767,A -85,B 0,C 180,E1 30426.647,E2 30426.647} C_VEL
LIN {X 0,Y 176.881,Z 1240.756,A -85,B 0,C 180,E1 30437.618,E2 30437.618} C_VEL
LIN {X 0,Y 121.074,Z 1265.166,A -85,B 0,C 180,E1 30461.211,E2 30461.211} C_VEL
LIN {X 0,Y 99.407,Z 1274.565,A -85,B 0,C 180,E1 30496.76,E2 30496.76} C_VEL
LIN {X 0,Y 98.902,Z 1275.091,A -85,B 0,C 180,E1 30514.404,E2 30514.404} C_VEL
LIN {X 0,Y 110.241,Z 1269.542,A -85,B 0,C 180,E1 30548.297,E2 30548.297} C_VEL
LIN {X 0,Y 159.327,Z 1249.19,A -85,B 0,C 180,E1 30577.382,E2 30577.382} C_VEL
LIN {X 0,Y 225.727,Z 1213.651,A -85,B 0,C 180,E1 30591.426,E2 30591.426} C_VEL
LIN {X 0,Y 291.827,Z 1164.607,A -85,B 0,C 180,E1 30598.336,E2 30598.336} C_VEL
LIN {X 0,Y 304.666,Z 1152.914,A -85,B 0,C 180,E1 30599.468,E2 30599.468} C_VEL
LIN {X 0,Y 304.254,Z 1153.023,A -85,B 0,C 180,E1 30601.704,E2 30601.704} C_VEL
LIN {X 0,Y 241.075,Z 1202.151,A -85,B 0,C 180,E1 30607.963,E2 30607.963} C_VEL
LIN {X 0,Y 176.455,Z 1238.065,A -85,B 0,C 180,E1 30619.42,E2 30619.42} C_VEL
LIN {X 0,Y 121.185,Z 1260.458,A -85,B 0,C 180,E1 30643.234,E2 30643.234} C_VEL
LIN {X 0,Y 99.797,Z 1268.219,A -85,B 0,C 180,E1 30676.807,E2 30676.807} C_VEL
LIN {X 0,Y 99.826,Z 1268.194,A -85,B 0,C 180,E1 30703.183,E2 30703.183} C_VEL
LIN {X 0,Y 127.109,Z 1258.338,A -85,B 0,C 180,E1 30740.922,E2 30740.922} C_VEL
LIN {X 0,Y 183.358,Z 1234.715,A -85,B 0,C 180,E1 30762.198,E2 30762.198} C_VEL
LIN {X 0,Y 197.144,Z 1227.732,A -85,B 0,C 180,E1 30765.171,E2 30765.171} C_VEL
LIN {X 0,Y 220.588,Z 1214.214,A -85,B 0,C 180,E1 30771.493,E2 30771.493} C_VEL
LIN {X 0,Y 286.875,Z 1168.005,A -85,B 0,C 180,E1 30778.362,E2 30778.362} C_VEL
LIN {X 0,Y 298.68,Z 1158.005,A -85,B 0,C 180,E1 30779.394,E2 30779.394} C_VEL
LIN {X 0,Y 232.522,Z 1208.401,A -85,B 0,C 180,E1 30785.481,E2 30785.481} C_VEL
LIN {X 0,Y 163.342,Z 1245.714,A -85,B 0,C 180,E1 30797.712,E2 30797.712} C_VEL
LIN {X 0,Y 108.418,Z 1267.634,A -85,B 0,C 180,E1 30824.152,E2 30824.152} C_VEL
LIN {X 0,Y 91.514,Z 1274.298,A -85,B 0,C 180,E1 30855.594,E2 30855.594} C_VEL
LIN {X 0,Y 90.872,Z 1274.826,A -85,B 0,C 180,E1 30874.794,E2 30874.794} C_VEL
LIN {X 0,Y 103.86,Z 1269.271,A -85,B 0,C 180,E1 30911.133,E2 30911.133} C_VEL
LIN {X 0,Y 154.64,Z 1249.642,A -85,B 0,C 180,E1 30939.745,E2 30939.745} C_VEL
LIN {X 0,Y 221.703,Z 1215.174,A -85,B 0,C 180,E1 30953.175,E2 30953.175} C_VEL
LIN {X 0,Y 288.293,Z 1167.264,A -85,B 0,C 180,E1 30959.716,E2 30959.716} C_VEL
LIN {X 0,Y 298.693,Z 1158.258,A -85,B 0,C 180,E1 30960.568,E2 30960.568} C_VEL
LIN {X 0,Y 232.738,Z 1207.137,A -85,B 0,C 180,E1 30966.858,E2 30966.858} C_VEL
LIN {X 0,Y 164.493,Z 1242.475,A -85,B 0,C 180,E1 30979.106,E2 30979.106} C_VEL
LIN {X 0,Y 108.895,Z 1262.938,A -85,B 0,C 180,E1 31005.805,E2 31005.805} C_VEL
LIN {X 0,Y 91.03,Z 1268.878,A -85,B 0,C 180,E1 31045.214,E2 31045.214} C_VEL
LIN {X 0,Y 94.587,Z 1267.507,A -85,B 0,C 180,E1 31073.653,E2 31073.653} C_VEL
LIN {X 0,Y 130.724,Z 1255.51,A -85,B 0,C 180,E1 31108.739,E2 31108.739} C_VEL
LIN {X 0,Y 194.442,Z 1228.373,A -85,B 0,C 180,E1 31127.401,E2 31127.401} C_VEL
LIN {X 0,Y 220.588,Z 1214.214,A -85,B 0,C 180,E1 31131.493,E2 31131.493} C_VEL
LIN {X 0,Y 245.334,Z 1198.681,A -85,B 0,C 180,E1 31136.479,E2 31136.479} C_VEL
LIN {X 0,Y 275.567,Z 1177.154,A -85,B 0,C 180,E1 31139.164,E2 31139.164} C_VEL
LIN {X 0,Y 210.009,Z 1221.049,A -85,B 0,C 180,E1 31146.057,E2 31146.057} C_VEL
LIN {X 0,Y 141.634,Z 1253.422,A -85,B 0,C 180,E1 31160.407,E2 31160.407} C_VEL
LIN {X 0,Y 91.208,Z 1271.179,A -85,B 0,C 180,E1 31194.373,E2 31194.373} C_VEL
LIN {X 0,Y 82.954,Z 1274.561,A -85,B 0,C 180,E1 31224.753,E2 31224.753} C_VEL
LIN {X 0,Y 86.396,Z 1272.918,A -85,B 0,C 180,E1 31256.062,E2 31256.062} C_VEL
LIN {X 0,Y 126.78,Z 1259.099,A -85,B 0,C 180,E1 31293.912,E2 31293.912} C_VEL
LIN {X 0,Y 191.986,Z 1230.84,A -85,B 0,C 180,E1 31311.284,E2 31311.284} C_VEL
LIN {X 0,Y 260.005,Z 1189.176,A -85,B 0,C 180,E1 31319.243,E2 31319.243} C_VEL
LIN {X 0,Y 275.36,Z 1177.536,A -85,B 0,C 180,E1 31320.795,E2 31320.795} C_VEL
LIN {X 0,Y 206.936,Z 1221.521,A -85,B 0,C 180,E1 31327.944,E2 31327.944} C_VEL
LIN {X 0,Y 139.859,Z 1251.239,A -85,B 0,C 180,E1 31342.68,E2 31342.68} C_VEL
LIN {X 0,Y 92.217,Z 1266.303,A -85,B 0,C 180,E1 31374.814,E2 31374.814} C_VEL
LIN {X 0,Y 83.02,Z 1269.142,A -85,B 0,C 180,E1 31404.751,E2 31404.751} C_VEL
LIN {X 0,Y 87.186,Z 1267.775,A -85,B 0,C 180,E1 31435.802,E2 31435.802} C_VEL
LIN {X 0,Y 125.839,Z 1256.039,A -85,B 0,C 180,E1 31471.604,E2 31471.604} C_VEL
LIN {X 0,Y 190.252,Z 1229.883,A -85,B 0,C 180,E1 31489.389,E2 31489.389} C_VEL
LIN {X 0,Y 245.334,Z 1198.681,A -85,B 0,C 180,E1 31496.479,E2 31496.479} C_VEL
LIN {X 0,Y 242.592,Z 1200.506,A -85,B 0,C 180,E1 31498.839,E2 31498.839} C_VEL
LIN {X 0,Y 223.928,Z 1212.339,A -85,B 0,C 180,E1 31502.08,E2 31502.08} C_VEL
LIN {X 0,Y 152.2,Z 1247.924,A -85,B 0,C 180,E1 31513.472,E2 31513.472} C_VEL
LIN {X 0,Y 92.045,Z 1268.693,A -85,B 0,C 180,E1 31542.086,E2 31542.086} C_VEL
LIN {X 0,Y 74.92,Z 1274.296,A -85,B 0,C 180,E1 31584.189,E2 31584.189} C_VEL
LIN {X 0,Y 79.983,Z 1272.409,A -85,B 0,C 180,E1 31620.79,E2 31620.79} C_VEL
LIN {X 0,Y 123.295,Z 1258.823,A -85,B 0,C 180,E1 31657.443,E2 31657.443} C_VEL
LIN {X 0,Y 190.883,Z 1230.563,A -85,B 0,C 180,E1 31673.806,E2 31673.806} C_VEL
LIN {X 0,Y 253.329,Z 1193.63,A -85,B 0,C 180,E1 31680.769,E2 31680.769} C_VEL
LIN {X 0,Y 184.303,Z 1232.477,A -85,B 0,C 180,E1 31688.819,E2 31688.819} C_VEL
LIN {X 0,Y 119.203,Z 1257.312,A -85,B 0,C 180,E1 31706.22,E2 31706.22} C_VEL
LIN {X 0,Y 79.88,Z 1268.067,A -85,B 0,C 180,E1 31741.629,E2 31741.629} C_VEL
LIN {X 0,Y 75.131,Z 1269.394,A -85,B 0,C 180,E1 31775.795,E2 31775.795} C_VEL
LIN {X 0,Y 97.647,Z 1263.471,A -85,B 0,C 180,E1 31820.706,E2 31820.706} C_VEL
LIN {X 0,Y 160.158,Z 1242.802,A -85,B 0,C 180,E1 31846.461,E2 31846.461} C_VEL
LIN {X 0,Y 229.972,Z 1208.303,A -85,B 0,C 180,E1 31856.969,E2 31856.969} C_VEL
LIN {X 0,Y 253.412,Z 1193.396,A -85,B 0,C 180,E1 31859.409,E2 31859.409} C_VEL
LIN {X 0,Y 223.928,Z 1212.339,A -85,B 0,C 180,E1 31862.08,E2 31862.08} C_VEL
LIN {X 0,Y 192.827,Z 1228.889,A -85,B 0,C 180,E1 31863.352,E2 31863.352} C_VEL
LIN {X 0,Y 120.357,Z 1258.491,A -85,B 0,C 180,E1 31878.92,E2 31878.92} C_VEL
LIN {X 0,Y 72.027,Z 1272.364,A -85,B 0,C 180,E1 31918.206,E2 31918.206} C_VEL
LIN {X 0,Y 66.827,Z 1274.033,A -85,B 0,C 180,E1 31956.526,E2 31956.526} C_VEL
LIN {X 0,Y 86.621,Z 1268.453,A -85,B 0,C 180,E1 32002.066,E2 32002.066} C_VEL
LIN {X 0,Y 150.517,Z 1247.745,A -85,B 0,C 180,E1 32029.55,E2 32029.55} C_VEL
LIN {X 0,Y 224.448,Z 1211.828,A -85,B 0,C 180,E1 32040.104,E2 32040.104} C_VEL
LIN {X 0,Y 230.369,Z 1208.356,A -85,B 0,C 180,E1 32040.788,E2 32040.788} C_VEL
LIN {X 0,Y 161.789,Z 1241.913,A -85,B 0,C 180,E1 32049.845,E2 32049.845} C_VEL
LIN {X 0,Y 94.393,Z 1263.383,A -85,B 0,C 180,E1 32073.914,E2 32073.914} C_VEL
LIN {X 0,Y 68.672,Z 1269.281,A -85,B 0,C 180,E1 32110.63,E2 32110.63} C_VEL
LIN {X 0,Y 68.701,Z 1269.257,A -85,B 0,C 180,E1 32149.354,E2 32149.354} C_VEL
LIN {X 0,Y 109.25,Z 1259.431,A -85,B 0,C 180,E1 32194.58,E2 32194.58} C_VEL
LIN {X 0,Y 179.637,Z 1234.294,A -85,B 0,C 180,E1 32213.182,E2 32213.182} C_VEL
LIN {X 0,Y 230.888,Z 1207.896,A -85,B 0,C 180,E1 32219.148,E2 32219.148} C_VEL
LIN {X 0,Y 192.827,Z 1228.889,A -85,B 0,C 180,E1 32223.352,E2 32223.352} C_VEL
LIN {X 0,Y 160.638,Z 1242.946,A -85,B 0,C 180,E1 32225.154,E2 32225.154} C_VEL
LIN {X 0,Y 92.706,Z 1265.435,A -85,B 0,C 180,E1 32245.761,E2 32245.761} C_VEL
LIN {X 0,Y 60.524,Z 1273.229,A -85,B 0,C 180,E1 32287.903,E2 32287.903} C_VEL
LIN {X 0,Y 58.809,Z 1273.768,A -85,B 0,C 180,E1 32317.42,E2 32317.42} C_VEL
LIN {X 0,Y 81.761,Z 1268.179,A -85,B 0,C 180,E1 32366.679,E2 32366.679} C_VEL
LIN {X 0,Y 149.111,Z 1247.512,A -85,B 0,C 180,E1 32392.706,E2 32392.706} C_VEL
LIN {X 0,Y 204.982,Z 1222.335,A -85,B 0,C 180,E1 32401.013,E2 32401.013} C_VEL
LIN {X 0,Y 132.253,Z 1252.056,A -85,B 0,C 180,E1 32412.646,E2 32412.646} C_VEL
LIN {X 0,Y 73.506,Z 1267.109,A -85,B 0,C 180,E1 32443.704,E2 32443.704} C_VEL
LIN {X 0,Y 59.037,Z 1269.934,A -85,B 0,C 180,E1 32482.608,E2 32482.608} C_VEL
LIN {X 0,Y 69.079,Z 1267.969,A -85,B 0,C 180,E1 32530.324,E2 32530.324} C_VEL
LIN {X 0,Y 125.234,Z 1254.266,A -85,B 0,C 180,E1 32565.325,E2 32565.325} C_VEL
LIN {X 0,Y 197.116,Z 1226.188,A -85,B 0,C 180,E1 32578.062,E2 32578.062} C_VEL
LIN {X 0,Y 207.733,Z 1220.802,A -85,B 0,C 180,E1 32579.219,E2 32579.219} C_VEL
LIN {X 0,Y 160.638,Z 1242.946,A -85,B 0,C 180,E1 32585.154,E2 32585.154} C_VEL
LIN {X 0,Y 127.745,Z 1254.27,A -85,B 0,C 180,E1 32587.977,E2 32587.977} C_VEL
LIN {X 0,Y 67.124,Z 1270.09,A -85,B 0,C 180,E1 32617.673,E2 32617.673} C_VEL
LIN {X 0,Y 50.895,Z 1273.501,A -85,B 0,C 180,E1 32661.428,E2 32661.428} C_VEL
LIN {X 0,Y 58.661,Z 1271.839,A -85,B 0,C 180,E1 32710.321,E2 32710.321} C_VEL
LIN {X 0,Y 115.96,Z 1257.993,A -85,B 0,C 180,E1 32749.088,E2 32749.088} C_VEL
LIN {X 0,Y 182.119,Z 1233.343,A -85,B 0,C 180,E1 32760.603,E2 32760.603} C_VEL
LIN {X 0,Y 109.856,Z 1258.294,A -85,B 0,C 180,E1 32774.675,E2 32774.675} C_VEL
LIN {X 0,Y 59.534,Z 1268.868,A -85,B 0,C 180,E1 32810.389,E2 32810.389} C_VEL
LIN {X 0,Y 51.179,Z 1270.187,A -85,B 0,C 180,E1 32858.524,E2 32858.524} C_VEL
LIN {X 0,Y 82.794,Z 1264.551,A -85,B 0,C 180,E1 32913.073,E2 32913.073} C_VEL
LIN {X 0,Y 151.789,Z 1245.188,A -85,B 0,C 180,E1 32934.707,E2 32934.707} C_VEL
LIN {X 0,Y 182.195,Z 1233.186,A -85,B 0,C 180,E1 32939.424,E2 32939.424} C_VEL
LIN {X 0,Y 127.745,Z 1254.27,A -85,B 0,C 180,E1 32947.977,E2 32947.977} C_VEL
LIN {X 0,Y 94.499,Z 1263.005,A -85,B 0,C 180,E1 32952.757,E2 32952.757} C_VEL
LIN {X 0,Y 45.84,Z 1272.693,A -85,B 0,C 180,E1 33000.22,E2 33000.22} C_VEL
LIN {X 0,Y 42.85,Z 1273.239,A -85,B 0,C 180,E1 33040.21,E2 33040.21} C_VEL
LIN {X 0,Y 80.23,Z 1266.346,A -85,B 0,C 180,E1 33101.112,E2 33101.112} C_VEL
LIN {X 0,Y 154.94,Z 1244.394,A -85,B 0,C 180,E1 33120.169,E2 33120.169} C_VEL
LIN {X 0,Y 159.429,Z 1242.731,A -85,B 0,C 180,E1 33120.953,E2 33120.953} C_VEL
LIN {X 0,Y 87.584,Z 1263.3,A -85,B 0,C 180,E1 33137.563,E2 33137.563} C_VEL
LIN {X 0,Y 46.417,Z 1270.079,A -85,B 0,C 180,E1 33180.614,E2 33180.614} C_VEL
LIN {X 0,Y 43.221,Z 1270.452,A -85,B 0,C 180,E1 33220.109,E2 33220.109} C_VEL
LIN {X 0,Y 79.391,Z 1264.823,A -85,B 0,C 180,E1 33278.403,E2 33278.403} C_VEL
LIN {X 0,Y 154.312,Z 1244.402,A -85,B 0,C 180,E1 33298.281,E2 33298.281} C_VEL
LIN {X 0,Y 159.414,Z 1242.635,A -85,B 0,C 180,E1 33299.195,E2 33299.195} C_VEL
LIN {X 0,Y 94.499,Z 1263.005,A -85,B 0,C 180,E1 33312.757,E2 33312.757} C_VEL
LIN {X 0,Y 61.751,Z 1269.042,A -85,B 0,C 180,E1 33322.103,E2 33322.103} C_VEL
LIN {X 0,Y 34.967,Z 1272.969,A -85,B 0,C 180,E1 33377.47,E2 33377.47} C_VEL
LIN {X 0,Y 47.305,Z 1271.298,A -85,B 0,C 180,E1 33443.359,E2 33443.359} C_VEL
LIN {X 0,Y 113.979,Z 1257.443,A -85,B 0,C 180,E1 33477.415,E2 33477.415} C_VEL
LIN {X 0,Y 135.116,Z 1251.103,A -85,B 0,C 180,E1 33480.832,E2 33480.832} C_VEL
LIN {X 0,Y 71.874,Z 1265.977,A -85,B 0,C 180,E1 33498.094,E2 33498.094} C_VEL
LIN {X 0,Y 35.217,Z 1270.726,A -85,B 0,C 180,E1 33557.546,E2 33557.546} C_VEL
LIN {X 0,Y 48.136,Z 1269.38,A -85,B 0,C 180,E1 33622.032,E2 33622.032} C_VEL
LIN {X 0,Y 114.213,Z 1256.909,A -85,B 0,C 180,E1 33655.457,E2 33655.457} C_VEL
LIN {X 0,Y 135.261,Z 1250.964,A -85,B 0,C 180,E1 33659.044,E2 33659.044} C_VEL
LIN {X 0,Y 61.751,Z 1269.042,A -85,B 0,C 180,E1 33682.103,E2 33682.103} C_VEL
LIN {X 0,Y 32.168,Z 1272.192,A -85,B 0,C 180,E1 33707.31,E2 33707.31} C_VEL
LIN {X 0,Y 27.061,Z 1272.707,A -85,B 0,C 180,E1 33766.3,E2 33766.3} C_VEL
LIN {X 0,Y 69.292,Z 1267.087,A -85,B 0,C 180,E1 33830.393,E2 33830.393} C_VEL
LIN {X 0,Y 107.592,Z 1258.833,A -85,B 0,C 180,E1 33840.617,E2 33840.617} C_VEL
LIN {X 0,Y 56.07,Z 1268.187,A -85,B 0,C 180,E1 33858.61,E2 33858.61} C_VEL
LIN {X 0,Y 27.396,Z 1270.991,A -85,B 0,C 180,E1 33913.905,E2 33913.905} C_VEL
LIN {X 0,Y 43.59,Z 1269.649,A -85,B 0,C 180,E1 33990.525,E2 33990.525} C_VEL
LIN {X 0,Y 103.309,Z 1259.778,A -85,B 0,C 180,E1 34017.816,E2 34017.816} C_VEL
LIN {X 0,Y 107.801,Z 1258.712,A -85,B 0,C 180,E1 34019.432,E2 34019.432} C_VEL
LIN {X 0,Y 42.929,Z 1271.012,A -85,B 0,C 180,E1 34047.873,E2 34047.873} C_VEL
LIN {X 0,Y 32.168,Z 1272.192,A -85,B 0,C 180,E1 34067.31,E2 34067.31} C_VEL
LIN {X 0,Y 21.515,Z 1272.24,A -85,B 0,C 180,E1 34148.249,E2 34148.249} C_VEL
LIN {X 0,Y 83.516,Z 1264.115,A -85,B 0,C 180,E1 34201.072,E2 34201.072} C_VEL
LIN {X 0,Y 27.879,Z 1270.878,A -85,B 0,C 180,E1 34235.218,E2 34235.218} C_VEL
LIN {X 0,Y 19.848,Z 1271.246,A -85,B 0,C 180,E1 34312.47,E2 34312.47} C_VEL
LIN {X 0,Y 75.997,Z 1265.326,A -85,B 0,C 180,E1 34377.119,E2 34377.119} C_VEL
LIN {X 0,Y 83.506,Z 1264.059,A -85,B 0,C 180,E1 34378.951,E2 34378.951} C_VEL
LIN {X 0,Y 25.777,Z 1271.974,A -85,B 0,C 180,E1 34417.568,E2 34417.568} C_VEL
LIN {X 0,Y 21.515,Z 1272.24,A -85,B 0,C 180,E1 34508.249,E2 34508.249} C_VEL
LIN {X 0,Y 45.221,Z 1269.659,A -85,B 0,C 180,E1 34558.099,E2 34558.099} C_VEL
LIN {X 0,Y 53.158,Z 1268.726,A -85,B 0,C 180,E1 34561.562,E2 34561.562} C_VEL
LIN {X 0,Y 12.697,Z 1271.521,A -85,B 0,C 180,E1 34613.262,E2 34613.262} C_VEL
LIN {X 0,Y 38.287,Z 1270.186,A -85,B 0,C 180,E1 34732.37,E2 34732.37} C_VEL
LIN {X 0,Y 53.133,Z 1268.722,A -85,B 0,C 180,E1 34739.354,E2 34739.354} C_VEL
LIN {X 0,Y 12.411,Z 1272.171,A -85,B 0,C 180,E1 34792.322,E2 34792.322} C_VEL
LIN {X 0,Y 23.846,Z 1271.637,A -85,B 0,C 180,E1 34902.771,E2 34902.771} C_VEL
LIN {X 0,Y 45.221,Z 1269.659,A -85,B 0,C 180,E1 34918.099,E2 34918.099} C_VEL
LIN {X 0,Y 20.965,Z 1271.469,A -85,B 0,C 180,E1 34925.388,E2 34925.388} C_VEL
LIN {X 0,Y 6.708,Z 1271.785,A -85,B 0,C 180,E1 34938.309,E2 34938.309} C_VEL
LIN {X 0,Y 18.34,Z 1271.599,A -85,B 0,C 180,E1 35099.517,E2 35099.517} C_VEL
LIN {X 0,Y 18.196,Z 1271.608,A -85,B 0,C 180,E1 34920.566,E2 34920.566} C_VEL
LIN {X 0,Y 6.708,Z 1271.785,A -85,B 0,C 180,E1 34938.309,E2 34938.309} C_VEL
LIN {X 0,Y 4.856,Z 1273.785,A -85,B 0,C 180,E1 34945.918,E2 34945.918} C_VEL
LIN {X 0,Y 4.856,Z 1292,A -85,B 0,C 180,E1 34945.918,E2 34945.918} C_VEL
LIN {X 0,Y 4.856,Z 1292,A -85,B 0,C 180,E1 34945.918,E2 34945.918}

QRS_NEXT_CUT()
PTP {E1 35097.077,E2 35097.077}
PTP {X 0,Y 759.921,A -85,B 0,C 180,E1 35097.077,E2 35097.077,E3 0,E4 0,E5 0,E6 0}
QRS_SPEED_INIT()
LIN {X 0,Y 759.921,Z 1292,A -85,B 0,C 180,E1 35097.077,E2 35097.077,E3 0,E4 0,E5 0,E6 0} C_VEL
LIN {X 0,Y 759.921,Z 396.653,A -85,B 0,C 180,E1 35097.077,E2 35097.077} C_VEL
LIN {X 0,Y 759.921,Z 388.573,A -85,B 0,C 180,E1 35097.077,E2 35097.077} C_VEL
LIN {X 0,Y 759.919,Z 386.573,A -85,B 0,C 180,E1 35096.926,E2 35096.926} C_VEL
LIN {X 0,Y 759.83,Z 386.574,A -85,B 0,C 180,E1 35094.184,E2 35094.184} C_VEL
LIN {X 0,Y 759.825,Z 386.574,A -85,B 0,C 180,E1 35091.829,E2 35091.829} C_VEL
LIN {X 0,Y 759.841,Z 386.575,A -85,B 0,C 180,E1 35089.46,E2 35089.46} C_VEL
LIN {X 0,Y 759.918,Z 386.57,A -85,B 0,C 180,E1 35086.61,E2 35086.61} C_VEL
LIN {X 0,Y 759.844,Z 386.572,A -85,B 0,C 180,E1 35083.879,E2 35083.879} C_VEL
LIN {X 0,Y 759.843,Z 386.574,A -85,B 0,C 180,E1 35081.431,E2 35081.431} C_VEL
LIN {X 0,Y 759.916,Z 386.577,A -85,B 0,C 180,E1 35078.706,E2 35078.706} C_VEL
LIN {X 0,Y 759.868,Z 386.569,A -85,B 0,C 180,E1 35075.843,E2 35075.843} C_VEL
LIN {X 0,Y 759.853,Z 386.572,A -85,B 0,C 180,E1 35073.301,E2 35073.301} C_VEL
LIN {X 0,Y 759.907,Z 386.578,A -85,B 0,C 180,E1 35070.607,E2 35070.607} C_VEL
LIN {X 0,Y 759.879,Z 386.568,A -85,B 0,C 180,E1 35067.618,E2 35067.618} C_VEL
LIN {X 0,Y 759.868,Z 386.572,A -85,B 0,C 180,E1 35064.921,E2 35064.921} C_VEL
LIN {X 0,Y 759.906,Z 386.571,A -85,B 0,C 180,E1 35062.127,E2 35062.127} C_VEL
LIN {X 0,Y 759.879,Z 386.568,A -85,B 0,C 180,E1 35059.273,E2 35059.273} C_VEL
LIN {X 0,Y 759.9,Z 386.576,A -85,B 0,C 180,E1 35056.462,E2 35056.462} C_VEL
LIN {X 0,Y 759.916,Z 386.565,A -85,B 0,C 180,E1 35053.421,E2 35053.421} C_VEL
LIN {X 0,Y 759.902,Z 386.602,A -85,B 0,C 180,E1 35051.635,E2 35051.635} C_VEL
LIN {X 0,Y 759.88,Z 398.346,A -85,B 0,C 180,E1 35050.866,E2 35050.866} C_VEL
LIN {X 0,Y 759.912,Z 608.567,A -85,B 0,C 180,E1 35048.336,E2 35048.336} C_VEL
LIN {X 0,Y 759.916,Z 833.718,A -85,B 0,C 180,E1 35045.723,E2 35045.723} C_VEL
LIN {X 0,Y 759.918,Z 877.059,A -85,B 0,C 180,E1 35045.204,E2 35045.204} C_VEL
LIN {X 0,Y 759.907,Z 902.512,A -85,B 0,C 180,E1 35044.767,E2 35044.767} C_VEL
LIN {X 0,Y 759.908,Z 929.633,A -85,B 0,C 180,E1 35044.142,E2 35044.142} C_VEL
LIN {X 0,Y 759.909,Z 951.796,A -85,B 0,C 180,E1 35043.503,E2 35043.503} C_VEL
LIN {X 0,Y 759.919,Z 969.721,A -85,B 0,C 180,E1 35042.91,E2 35042.91} C_VEL
LIN {X 0,Y 759.919,Z 988.329,A -85,B 0,C 180,E1 35042.215,E2 35042.215} C_VEL
LIN {X 0,Y 759.912,Z 1007.779,A -85,B 0,C 180,E1 35041.397,E2 35041.397} C_VEL
LIN {X 0,Y 759.914,Z 1026.488,A -85,B 0,C 180,E1 35040.518,E2 35040.518} C_VEL
LIN {X 0,Y 759.906,Z 1045.694,A -85,B 0,C 180,E1 35039.517,E2 35039.517} C_VEL
LIN {X 0,Y 759.916,Z 1068.899,A -85,B 0,C 180,E1 35038.166,E2 35038.166} C_VEL
LIN {X 0,Y 759.917,Z 1089.261,A -85,B 0,C 180,E1 35036.823,E2 35036.823} C_VEL
LIN {X 0,Y 759.914,Z 1106.63,A -85,B 0,C 180,E1 35035.562,E2 35035.562} C_VEL
LIN {X 0,Y 759.891,Z 1126.398,A -85,B 0,C 180,E1 35033.986,E2 35033.986} C_VEL
LIN {X 0,Y 759.901,Z 1144.729,A -85,B 0,C 180,E1 35032.328,E2 35032.328} C_VEL
LIN {X 0,Y 759.907,Z 1159.22,A -85,B 0,C 180,E1 35030.886,E2 35030.886} C_VEL
LIN {X 0,Y 759.917,Z 1175.276,A -85,B 0,C 180,E1 35029.12,E2 35029.12} C_VEL
LIN {X 0,Y 759.874,Z 1189.782,A -85,B 0,C 180,E1 35027.296,E2 35027.296} C_VEL
LIN {X 0,Y 759.886,Z 1200.938,A -85,B 0,C 180,E1 35025.723,E2 35025.723} C_VEL
LIN {X 0,Y 759.914,Z 1210.345,A -85,B 0,C 180,E1 35024.24,E2 35024.24} C_VEL
LIN {X 0,Y 759.917,Z 1219.071,A -85,B 0,C 180,E1 35022.689,E2 35022.689} C_VEL
LIN {X 0,Y 759.895,Z 1227.38,A -85,B 0,C 180,E1 35020.995,E2 35020.995} C_VEL
LIN {X 0,Y 759.867,Z 1235.603,A -85,B 0,C 180,E1 35019.005,E2 35019.005} C_VEL
LIN {X 0,Y 759.907,Z 1242.451,A -85,B 0,C 180,E1 35016.873,E2 35016.873} C_VEL
LIN {X 0,Y 759.915,Z 1247.108,A -85,B 0,C 180,E1 35014.903,E2 35014.903} C_VEL
LIN {X 0,Y 759.911,Z 1250.245,A -85,B 0,C 180,E1 35012.925,E2 35012.925} C_VEL
LIN {X 0,Y 759.875,Z 1251.703,A -85,B 0,C 180,E1 35010.977,E2 35010.977} C_VEL
LIN {X 0,Y 759.864,Z 1251.839,A -85,B 0,C 180,E1 35009.393,E2 35009.393} C_VEL
LIN {X 0,Y 759.91,Z 1250.983,A -85,B 0,C 180,E1 35007.81,E2 35007.81} C_VEL
LIN {X 0,Y 759.914,Z 1248.872,A -85,B 0,C 180,E1 35005.998,E2 35005.998} C_VEL
LIN {X 0,Y 759.916,Z 1244.651,A -85,B 0,C 180,E1 35003.879,E2 35003.879} C_VEL
LIN {X 0,Y 759.895,Z 1239.212,A -85,B 0,C 180,E1 35001.979,E2 35001.979} C_VEL
LIN {X 0,Y 759.887,Z 1232.904,A -85,B 0,C 180,E1 35000.224,E2 35000.224} C_VEL
LIN {X 0,Y 759.907,Z 1226.336,A -85,B 0,C 180,E1 34998.691,E2 34998.691} C_VEL
LIN {X 0,Y 759.91,Z 1218.691,A -85,B 0,C 180,E1 34997.149,E2 34997.149} C_VEL
LIN {X 0,Y 759.916,Z 1209.709,A -85,B 0,C 180,E1 34995.564,E2 34995.564} C_VEL
LIN {X 0,Y 759.887,Z 1198.736,A -85,B 0,C 180,E1 34993.857,E2 34993.857} C_VEL
LIN {X 0,Y 759.911,Z 1183.557,A -85,B 0,C 180,E1 34991.807,E2 34991.807} C_VEL
LIN {X 0,Y 759.88,Z 1170.329,A -85,B 0,C 180,E1 34990.232,E2 34990.232} C_VEL
LIN {X 0,Y 759.901,Z 1156.898,A -85,B 0,C 180,E1 34988.784,E2 34988.784} C_VEL
LIN {X 0,Y 759.906,Z 1139.432,A -85,B 0,C 180,E1 34987.076,E2 34987.076} C_VEL
LIN {X 0,Y 759.914,Z 1120.32,A -85,B 0,C 180,E1 34985.429,E2 34985.429} C_VEL
LIN {X 0,Y 759.897,Z 1103.29,A -85,B 0,C 180,E1 34984.095,E2 34984.095} C_VEL
LIN {X 0,Y 759.914,Z 1081.181,A -85,B 0,C 180,E1 34982.534,E2 34982.534} C_VEL
LIN {X 0,Y 759.908,Z 1060.687,A -85,B 0,C 180,E1 34981.252,E2 34981.252} C_VEL
LIN {X 0,Y 759.913,Z 1042.397,A -85,B 0,C 180,E1 34980.215,E2 34980.215} C_VEL
LIN {X 0,Y 759.912,Z 1023.885,A -85,B 0,C 180,E1 34979.264,E2 34979.264} C_VEL
LIN {X 0,Y 759.915,Z 1003.658,A -85,B 0,C 180,E1 34978.33,E2 34978.33} C_VEL
LIN {X 0,Y 759.918,Z 978.398,A -85,B 0,C 180,E1 34977.306,E2 34977.306} C_VEL
LIN {X 0,Y 759.907,Z 954.584,A -85,B 0,C 180,E1 34976.493,E2 34976.493} C_VEL
LIN {X 0,Y 759.907,Z 931.457,A -85,B 0,C 180,E1 34975.814,E2 34975.814} C_VEL
LIN {X 0,Y 759.907,Z 904.84,A -85,B 0,C 180,E1 34975.192,E2 34975.192} C_VEL
LIN {X 0,Y 759.912,Z 879.016,A -85,B 0,C 180,E1 34974.735,E2 34974.735} C_VEL
LIN {X 0,Y 759.917,Z 839.344,A -85,B 0,C 180,E1 34974.251,E2 34974.251} C_VEL
LIN {X 0,Y 759.91,Z 616.02,A -85,B 0,C 180,E1 34971.662,E2 34971.662} C_VEL
LIN {X 0,Y 759.886,Z 406.481,A -85,B 0,C 180,E1 34969.144,E2 34969.144} C_VEL
LIN {X 0,Y 759.888,Z 397.792,A -85,B 0,C 180,E1 34969.028,E2 34969.028} C_VEL
LIN {X 0,Y 759.893,Z 386.573,A -85,B 0,C 180,E1 34968.252,E2 34968.252} C_VEL
LIN {X 0,Y 759.903,Z 386.576,A -85,B 0,C 180,E1 34965.386,E2 34965.386} C_VEL
LIN {X 0,Y 759.907,Z 386.564,A -85,B 0,C 180,E1 34962.423,E2 34962.423} C_VEL
LIN {X 0,Y 759.905,Z 386.576,A -85,B 0,C 180,E1 34959.431,E2 34959.431} C_VEL
LIN {X 0,Y 759.891,Z 386.568,A -85,B 0,C 180,E1 34956.589,E2 34956.589} C_VEL
LIN {X 0,Y 759.892,Z 386.566,A -85,B 0,C 180,E1 34953.821,E2 34953.821} C_VEL
LIN {X 0,Y 759.91,Z 386.575,A -85,B 0,C 180,E1 34950.917,E2 34950.917} C_VEL
LIN {X 0,Y 759.919,Z 386.562,A -85,B 0,C 180,E1 34947.932,E2 34947.932} C_VEL
LIN {X 0,Y 759.905,Z 386.575,A -85,B 0,C 180,E1 34944.902,E2 34944.902} C_VEL
LIN {X 0,Y 759.897,Z 386.567,A -85,B 0,C 180,E1 34942.025,E2 34942.025} C_VEL
LIN {X 0,Y 759.888,Z 386.566,A -85,B 0,C 180,E1 34939.286,E2 34939.286} C_VEL
LIN {X 0,Y 759.911,Z 386.577,A -85,B 0,C 180,E1 34936.419,E2 34936.419} C_VEL
LIN {X 0,Y 759.912,Z 386.563,A -85,B 0,C 180,E1 34933.39,E2 34933.39} C_VEL
LIN {X 0,Y 759.894,Z 386.574,A -85,B 0,C 180,E1 34930.462,E2 34930.462} C_VEL
LIN {X 0,Y 759.897,Z 386.569,A -85,B 0,C 180,E1 34927.637,E2 34927.637} C_VEL
LIN {X 0,Y 759.886,Z 386.567,A -85,B 0,C 180,E1 34924.831,E2 34924.831} C_VEL
LIN {X 0,Y 759.91,Z 386.576,A -85,B 0,C 180,E1 34921.961,E2 34921.961} C_VEL
LIN {X 0,Y 759.906,Z 386.564,A -85,B 0,C 180,E1 34918.869,E2 34918.869} C_VEL
LIN {X 0,Y 759.885,Z 386.572,A -85,B 0,C 180,E1 34916.001,E2 34916.001} C_VEL
LIN {X 0,Y 759.9,Z 386.57,A -85,B 0,C 180,E1 34913.199,E2 34913.199} C_VEL
LIN {X 0,Y 759.886,Z 386.565,A -85,B 0,C 180,E1 34910.38,E2 34910.38} C_VEL
LIN {X 0,Y 759.899,Z 386.576,A -85,B 0,C 180,E1 34907.512,E2 34907.512} C_VEL
LIN {X 0,Y 759.916,Z 386.563,A -85,B 0,C 180,E1 34904.508,E2 34904.508} C_VEL
LIN {X 0,Y 759.871,Z 386.57,A -85,B 0,C 180,E1 34901.749,E2 34901.749} C_VEL
LIN {X 0,Y 759.911,Z 386.577,A -85,B 0,C 180,E1 34899.029,E2 34899.029} C_VEL
LIN {X 0,Y 759.894,Z 386.565,A -85,B 0,C 180,E1 34896.009,E2 34896.009} C_VEL
LIN {X 0,Y 759.873,Z 386.572,A -85,B 0,C 180,E1 34893.255,E2 34893.255} C_VEL
LIN {X 0,Y 759.908,Z 386.573,A -85,B 0,C 180,E1 34890.52,E2 34890.52} C_VEL
LIN {X 0,Y 759.882,Z 386.567,A -85,B 0,C 180,E1 34887.619,E2 34887.619} C_VEL
LIN {X 0,Y 759.874,Z 386.573,A -85,B 0,C 180,E1 34884.898,E2 34884.898} C_VEL
LIN {X 0,Y 759.907,Z 386.571,A -85,B 0,C 180,E1 34882.086,E2 34882.086} C_VEL
LIN {X 0,Y 759.873,Z 386.568,A -85,B 0,C 180,E1 34879.257,E2 34879.257} C_VEL
LIN {X 0,Y 759.872,Z 386.574,A -85,B 0,C 180,E1 34876.583,E2 34876.583} C_VEL
LIN {X 0,Y 759.908,Z 386.575,A -85,B 0,C 180,E1 34873.749,E2 34873.749} C_VEL
LIN {X 0,Y 759.915,Z 386.8,A -85,B 0,C 180,E1 34873.531,E2 34873.531} C_VEL
LIN {X 0,Y 759.904,Z 427.619,A -85,B 0,C 180,E1 34870.918,E2 34870.918} C_VEL
LIN {X 0,Y 759.911,Z 644.419,A -85,B 0,C 180,E1 34868.312,E2 34868.312} C_VEL
LIN {X 0,Y 759.917,Z 869.846,A -85,B 0,C 180,E1 34865.698,E2 34865.698} C_VEL
LIN {X 0,Y 759.917,Z 908.739,A -85,B 0,C 180,E1 34865.224,E2 34865.224} C_VEL
LIN {X 0,Y 759.907,Z 934.454,A -85,B 0,C 180,E1 34864.771,E2 34864.771} C_VEL
LIN {X 0,Y 759.907,Z 961.39,A -85,B 0,C 180,E1 34864.142,E2 34864.142} C_VEL
LIN {X 0,Y 759.908,Z 986.138,A -85,B 0,C 180,E1 34863.414,E2 34863.414} C_VEL
LIN {X 0,Y 759.918,Z 1013.047,A -85,B 0,C 180,E1 34862.471,E2 34862.471} C_VEL
LIN {X 0,Y 759.917,Z 1034.635,A -85,B 0,C 180,E1 34861.582,E2 34861.582} C_VEL
LIN {X 0,Y 759.909,Z 1053.68,A -85,B 0,C 180,E1 34860.701,E2 34860.701} C_VEL
LIN {X 0,Y 759.912,Z 1072.368,A -85,B 0,C 180,E1 34859.741,E2 34859.741} C_VEL
LIN {X 0,Y 759.906,Z 1090.653,A -85,B 0,C 180,E1 34858.705,E2 34858.705} C_VEL
LIN {X 0,Y 759.915,Z 1112.181,A -85,B 0,C 180,E1 34857.357,E2 34857.357} C_VEL
LIN {X 0,Y 759.898,Z 1133.579,A -85,B 0,C 180,E1 34855.839,E2 34855.839} C_VEL
LIN {X 0,Y 759.91,Z 1150.784,A -85,B 0,C 180,E1 34854.489,E2 34854.489} C_VEL
LIN {X 0,Y 759.91,Z 1169.82,A -85,B 0,C 180,E1 34852.842,E2 34852.842} C_VEL
LIN {X 0,Y 759.904,Z 1186.464,A -85,B 0,C 180,E1 34851.216,E2 34851.216} C_VEL
LIN {X 0,Y 759.88,Z 1199.93,A -85,B 0,C 180,E1 34849.768,E2 34849.768} C_VEL
LIN {X 0,Y 759.908,Z 1212.706,A -85,B 0,C 180,E1 34848.252,E2 34848.252} C_VEL
LIN {X 0,Y 759.898,Z 1227.01,A -85,B 0,C 180,E1 34846.357,E2 34846.357} C_VEL
LIN {X 0,Y 759.917,Z 1239.175,A -85,B 0,C 180,E1 34844.48,E2 34844.48} C_VEL
LIN {X 0,Y 759.894,Z 1248.041,A -85,B 0,C 180,E1 34842.929,E2 34842.929} C_VEL
LIN {X 0,Y 759.91,Z 1255.769,A -85,B 0,C 180,E1 34841.386,E2 34841.386} C_VEL
LIN {X 0,Y 759.902,Z 1262.418,A -85,B 0,C 180,E1 34839.852,E2 34839.852} C_VEL
LIN {X 0,Y 759.916,Z 1268.292,A -85,B 0,C 180,E1 34838.249,E2 34838.249} C_VEL
LIN {X 0,Y 759.917,Z 1273.753,A -85,B 0,C 180,E1 34836.425,E2 34836.425} C_VEL
LIN {X 0,Y 759.908,Z 1278.048,A -85,B 0,C 180,E1 34834.456,E2 34834.456} C_VEL
LIN {X 0,Y 759.903,Z 1280.672,A -85,B 0,C 180,E1 34832.492,E2 34832.492} C_VEL
LIN {X 0,Y 759.867,Z 1281.736,A -85,B 0,C 180,E1 34830.908,E2 34830.908} C_VEL
LIN {X 0,Y 759.863,Z 1281.828,A -85,B 0,C 180,E1 34829.4,E2 34829.4} C_VEL
LIN {X 0,Y 759.911,Z 1280.948,A -85,B 0,C 180,E1 34827.817,E2 34827.817} C_VEL
LIN {X 0,Y 759.913,Z 1278.809,A -85,B 0,C 180,E1 34826.005,E2 34826.005} C_VEL
LIN {X 0,Y 759.913,Z 1274.743,A -85,B 0,C 180,E1 34823.961,E2 34823.961} C_VEL
LIN {X 0,Y 759.888,Z 1269.34,A -85,B 0,C 180,E1 34822.062,E2 34822.062} C_VEL
LIN {X 0,Y 759.883,Z 1263.058,A -85,B 0,C 180,E1 34820.308,E2 34820.308} C_VEL
LIN {X 0,Y 759.906,Z 1256.517,A -85,B 0,C 180,E1 34818.775,E2 34818.775} C_VEL
LIN {X 0,Y 759.913,Z 1248.9,A -85,B 0,C 180,E1 34817.233,E2 34817.233} C_VEL
LIN {X 0,Y 759.915,Z 1240.149,A -85,B 0,C 180,E1 34815.683,E2 34815.683} C_VEL
LIN {X 0,Y 759.884,Z 1230.193,A -85,B 0,C 180,E1 34814.12,E2 34814.12} C_VEL
LIN {X 0,Y 759.89,Z 1217.146,A -85,B 0,C 180,E1 34812.302,E2 34812.302} C_VEL
LIN {X 0,Y 759.887,Z 1202.127,A -85,B 0,C 180,E1 34810.48,E2 34810.48} C_VEL
LIN {X 0,Y 759.902,Z 1188.095,A -85,B 0,C 180,E1 34808.953,E2 34808.953} C_VEL
LIN {X 0,Y 759.914,Z 1173.101,A -85,B 0,C 180,E1 34807.472,E2 34807.472} C_VEL
LIN {X 0,Y 759.899,Z 1152.4,A -85,B 0,C 180,E1 34805.643,E2 34805.643} C_VEL
LIN {X 0,Y 759.905,Z 1135.011,A -85,B 0,C 180,E1 34804.27,E2 34804.27} C_VEL
LIN {X 0,Y 759.913,Z 1116.276,A -85,B 0,C 180,E1 34802.924,E2 34802.924} C_VEL
LIN {X 0,Y 759.905,Z 1092.968,A -85,B 0,C 180,E1 34801.432,E2 34801.432} C_VEL
LIN {X 0,Y 759.91,Z 1074.119,A -85,B 0,C 180,E1 34800.353,E2 34800.353} C_VEL
LIN {X 0,Y 759.913,Z 1055.622,A -85,B 0,C 180,E1 34799.395,E2 34799.395} C_VEL
LIN {X 0,Y 759.913,Z 1036.804,A -85,B 0,C 180,E1 34798.515,E2 34798.515} C_VEL
LIN {X 0,Y 759.918,Z 1017.724,A -85,B 0,C 180,E1 34797.716,E2 34797.716} C_VEL
LIN {X 0,Y 759.919,Z 998.452,A -85,B 0,C 180,E1 34797,E2 34797} C_VEL
LIN {X 0,Y 759.913,Z 979.077,A -85,B 0,C 180,E1 34796.368,E2 34796.368} C_VEL
LIN {X 0,Y 759.91,Z 957.339,A -85,B 0,C 180,E1 34795.754,E2 34795.754} C_VEL
LIN {X 0,Y 759.907,Z 931.048,A -85,B 0,C 180,E1 34795.159,E2 34795.159} C_VEL
LIN {X 0,Y 759.913,Z 903.16,A -85,B 0,C 180,E1 34794.694,E2 34794.694} C_VEL
LIN {X 0,Y 759.907,Z 657.198,A -85,B 0,C 180,E1 34791.838,E2 34791.838} C_VEL
LIN {X 0,Y 759.897,Z 446.532,A -85,B 0,C 180,E1 34789.313,E2 34789.313} C_VEL
LIN {X 0,Y 759.905,Z 427.36,A -85,B 0,C 180,E1 34789.067,E2 34789.067} C_VEL
LIN {X 0,Y 759.914,Z 386.572,A -85,B 0,C 180,E1 34786.454,E2 34786.454} C_VEL
LIN {X 0,Y 759.87,Z 386.575,A -85,B 0,C 180,E1 34783.536,E2 34783.536} C_VEL
LIN {X 0,Y 759.855,Z 386.57,A -85,B 0,C 180,E1 34780.944,E2 34780.944} C_VEL
LIN {X 0,Y 759.917,Z 386.569,A -85,B 0,C 180,E1 34778.201,E2 34778.201} C_VEL
LIN {X 0,Y 759.856,Z 386.575,A -85,B 0,C 180,E1 34775.288,E2 34775.288} C_VEL
LIN {X 0,Y 759.84,Z 386.573,A -85,B 0,C 180,E1 34772.831,E2 34772.831} C_VEL
LIN {X 0,Y 759.876,Z 386.57,A -85,B 0,C 180,E1 34770.263,E2 34770.263} C_VEL
LIN {X 0,Y 759.862,Z 386.576,A -85,B 0,C 180,E1 34767.254,E2 34767.254} C_VEL
LIN {X 0,Y 759.827,Z 386.574,A -85,B 0,C 180,E1 34764.785,E2 34764.785} C_VEL
LIN {X 0,Y 759.829,Z 386.574,A -85,B 0,C 180,E1 34762.434,E2 34762.434} C_VEL
LIN {X 0,Y 759.914,Z 386.572,A -85,B 0,C 180,E1 34759.685,E2 34759.685} C_VEL
LIN {X 0,Y 759.829,Z 386.576,A -85,B 0,C 180,E1 34756.829,E2 34756.829} C_VEL
LIN {X 0,Y 759.813,Z 386.575,A -85,B 0,C 180,E1 34754.557,E2 34754.557} C_VEL
LIN {X 0,Y 759.807,Z 386.577,A -85,B 0,C 180,E1 34752.387,E2 34752.387} C_VEL
LIN {X 0,Y 759.806,Z 386.577,A -85,B 0,C 180,E1 34750.157,E2 34750.157} C_VEL
LIN {X 0,Y 759.818,Z 386.577,A -85,B 0,C 180,E1 34747.866,E2 34747.866} C_VEL
LIN {X 0,Y 759.88,Z 386.576,A -85,B 0,C 180,E1 34744.982,E2 34744.982} C_VEL
LIN {X 0,Y 759.816,Z 386.576,A -85,B 0,C 180,E1 34742.413,E2 34742.413} C_VEL
LIN {X 0,Y 759.812,Z 386.576,A -85,B 0,C 180,E1 34740.151,E2 34740.151} C_VEL
LIN {X 0,Y 759.815,Z 386.575,A -85,B 0,C 180,E1 34737.964,E2 34737.964} C_VEL
LIN {X 0,Y 759.919,Z 386.573,A -85,B 0,C 180,E1 34736.926,E2 34736.926} C_VEL
LIN {X 0,Y 758.933,Z 386.687,A -85,B 0,C 180,E1 34736.346,E2 34736.346} C_VEL
LIN {X 0,Y 752.464,Z 387.502,A -85,B 0,C 180,E1 34734.72,E2 34734.72} C_VEL
LIN {X 0,Y 751.9,Z 387.563,A -85,B 0,C 180,E1 34734.298,E2 34734.298} C_VEL
LIN {X 0,Y 751.886,Z 387.562,A -85,B 0,C 180,E1 34731.896,E2 34731.896} C_VEL
LIN {X 0,Y 751.9,Z 387.563,A -85,B 0,C 180,E1 34729.503,E2 34729.503} C_VEL
LIN {X 0,Y 751.978,Z 387.56,A -85,B 0,C 180,E1 34726.701,E2 34726.701} C_VEL
LIN {X 0,Y 751.909,Z 387.56,A -85,B 0,C 180,E1 34723.943,E2 34723.943} C_VEL
LIN {X 0,Y 751.904,Z 387.563,A -85,B 0,C 180,E1 34721.448,E2 34721.448} C_VEL
LIN {X 0,Y 751.976,Z 387.564,A -85,B 0,C 180,E1 34718.715,E2 34718.715} C_VEL
LIN {X 0,Y 751.925,Z 387.558,A -85,B 0,C 180,E1 34715.799,E2 34715.799} C_VEL
LIN {X 0,Y 751.917,Z 387.561,A -85,B 0,C 180,E1 34713.205,E2 34713.205} C_VEL
LIN {X 0,Y 751.975,Z 387.561,A -85,B 0,C 180,E1 34710.441,E2 34710.441} C_VEL
LIN {X 0,Y 751.939,Z 387.557,A -85,B 0,C 180,E1 34707.595,E2 34707.595} C_VEL
LIN {X 0,Y 751.929,Z 387.56,A -85,B 0,C 180,E1 34704.938,E2 34704.938} C_VEL
LIN {X 0,Y 751.968,Z 387.559,A -85,B 0,C 180,E1 34702.161,E2 34702.161} C_VEL
LIN {X 0,Y 751.942,Z 387.557,A -85,B 0,C 180,E1 34699.275,E2 34699.275} C_VEL
LIN {X 0,Y 751.965,Z 387.566,A -85,B 0,C 180,E1 34696.434,E2 34696.434} C_VEL
LIN {X 0,Y 751.967,Z 387.557,A -85,B 0,C 180,E1 34693.335,E2 34693.335} C_VEL
LIN {X 0,Y 751.982,Z 387.667,A -85,B 0,C 180,E1 34692.101,E2 34692.101} C_VEL
LIN {X 0,Y 753.239,Z 391.495,A -85,B 0,C 180,E1 34691.752,E2 34691.752} C_VEL
LIN {X 0,Y 753.309,Z 398.443,A -85,B 0,C 180,E1 34691.299,E2 34691.299} C_VEL
LIN {X 0,Y 753.815,Z 401.463,A -85,B 0,C 180,E1 34691.228,E2 34691.228} C_VEL
LIN {X 0,Y 753.625,Z 611.303,A -85,B 0,C 180,E1 34688.683,E2 34688.683} C_VEL
LIN {X 0,Y 753.412,Z 836.318,A -85,B 0,C 180,E1 34686.05,E2 34686.05} C_VEL
LIN {X 0,Y 753.359,Z 878.771,A -85,B 0,C 180,E1 34685.532,E2 34685.532} C_VEL
LIN {X 0,Y 753.27,Z 905.055,A -85,B 0,C 180,E1 34685.065,E2 34685.065} C_VEL
LIN {X 0,Y 753.182,Z 931.93,A -85,B 0,C 180,E1 34684.43,E2 34684.43} C_VEL
LIN {X 0,Y 753.092,Z 957.359,A -85,B 0,C 180,E1 34683.674,E2 34683.674} C_VEL
LIN {X 0,Y 752.955,Z 984.379,A -85,B 0,C 180,E1 34682.71,E2 34682.71} C_VEL
LIN {X 0,Y 752.859,Z 1005.809,A -85,B 0,C 180,E1 34681.815,E2 34681.815} C_VEL
LIN {X 0,Y 752.753,Z 1025.354,A -85,B 0,C 180,E1 34680.897,E2 34680.897} C_VEL
LIN {X 0,Y 752.662,Z 1044.904,A -85,B 0,C 180,E1 34679.873,E2 34679.873} C_VEL
LIN {X 0,Y 752.542,Z 1067.981,A -85,B 0,C 180,E1 34678.527,E2 34678.527} C_VEL
LIN {X 0,Y 752.423,Z 1089.27,A -85,B 0,C 180,E1 34677.111,E2 34677.111} C_VEL
LIN {X 0,Y 752.333,Z 1106.637,A -85,B 0,C 180,E1 34675.839,E2 34675.839} C_VEL
LIN {X 0,Y 752.236,Z 1126.496,A -85,B 0,C 180,E1 34674.237,E2 34674.237} C_VEL
LIN {X 0,Y 752.171,Z 1144.555,A -85,B 0,C 180,E1 34672.588,E2 34672.588} C_VEL
LIN {X 0,Y 752.103,Z 1159.227,A -85,B 0,C 180,E1 34671.113,E2 34671.113} C_VEL
LIN {X 0,Y 752.056,Z 1175.784,A -85,B 0,C 180,E1 34669.269,E2 34669.269} C_VEL
LIN {X 0,Y 751.969,Z 1189.787,A -85,B 0,C 180,E1 34667.484,E2 34667.484} C_VEL
LIN {X 0,Y 751.946,Z 1200.437,A -85,B 0,C 180,E1 34665.97,E2 34665.97} C_VEL
LIN {X 0,Y 751.959,Z 1210.349,A -85,B 0,C 180,E1 34664.394,E2 34664.394} C_VEL
LIN {X 0,Y 751.94,Z 1219.486,A -85,B 0,C 180,E1 34662.748,E2 34662.748} C_VEL
LIN {X 0,Y 751.911,Z 1228.098,A -85,B 0,C 180,E1 34660.958,E2 34660.958} C_VEL
LIN {X 0,Y 751.884,Z 1236.423,A -85,B 0,C 180,E1 34658.855,E2 34658.855} C_VEL
LIN {X 0,Y 751.91,Z 1242.67,A -85,B 0,C 180,E1 34656.87,E2 34656.87} C_VEL
LIN {X 0,Y 751.909,Z 1247.406,A -85,B 0,C 180,E1 34654.802,E2 34654.802} C_VEL
LIN {X 0,Y 751.917,Z 1250.369,A -85,B 0,C 180,E1 34652.817,E2 34652.817} C_VEL
LIN {X 0,Y 751.876,Z 1251.703,A -85,B 0,C 180,E1 34650.987,E2 34650.987} C_VEL
LIN {X 0,Y 751.864,Z 1251.839,A -85,B 0,C 180,E1 34649.387,E2 34649.387} C_VEL
LIN {X 0,Y 751.909,Z 1250.982,A -85,B 0,C 180,E1 34647.787,E2 34647.787} C_VEL
LIN {X 0,Y 751.915,Z 1248.871,A -85,B 0,C 180,E1 34645.955,E2 34645.955} C_VEL
LIN {X 0,Y 751.919,Z 1244.65,A -85,B 0,C 180,E1 34643.813,E2 34643.813} C_VEL
LIN {X 0,Y 751.913,Z 1238.954,A -85,B 0,C 180,E1 34641.817,E2 34641.817} C_VEL
LIN {X 0,Y 751.909,Z 1232.903,A -85,B 0,C 180,E1 34640.119,E2 34640.119} C_VEL
LIN {X 0,Y 751.929,Z 1225.977,A -85,B 0,C 180,E1 34638.491,E2 34638.491} C_VEL
LIN {X 0,Y 751.916,Z 1218.279,A -85,B 0,C 180,E1 34636.932,E2 34636.932} C_VEL
LIN {X 0,Y 751.947,Z 1208.977,A -85,B 0,C 180,E1 34635.284,E2 34635.284} C_VEL
LIN {X 0,Y 752.003,Z 1196.211,A -85,B 0,C 180,E1 34633.307,E2 34633.307} C_VEL
LIN {X 0,Y 752.031,Z 1182.202,A -85,B 0,C 180,E1 34631.442,E2 34631.442} C_VEL
LIN {X 0,Y 752.043,Z 1169.616,A -85,B 0,C 180,E1 34629.936,E2 34629.936} C_VEL
LIN {X 0,Y 752.117,Z 1155.334,A -85,B 0,C 180,E1 34628.39,E2 34628.39} C_VEL
LIN {X 0,Y 752.202,Z 1135.714,A -85,B 0,C 180,E1 34626.495,E2 34626.495} C_VEL
LIN {X 0,Y 752.284,Z 1119.297,A -85,B 0,C 180,E1 34625.079,E2 34625.079} C_VEL
LIN {X 0,Y 752.343,Z 1100.586,A -85,B 0,C 180,E1 34623.608,E2 34623.608} C_VEL
LIN {X 0,Y 752.473,Z 1078.829,A -85,B 0,C 180,E1 34622.087,E2 34622.087} C_VEL
LIN {X 0,Y 752.581,Z 1059.952,A -85,B 0,C 180,E1 34620.902,E2 34620.902} C_VEL
LIN {X 0,Y 752.669,Z 1041.586,A -85,B 0,C 180,E1 34619.855,E2 34619.855} C_VEL
LIN {X 0,Y 752.772,Z 1021.023,A -85,B 0,C 180,E1 34618.798,E2 34618.798} C_VEL
LIN {X 0,Y 752.931,Z 994.341,A -85,B 0,C 180,E1 34617.601,E2 34617.601} C_VEL
LIN {X 0,Y 753.026,Z 973.002,A -85,B 0,C 180,E1 34616.776,E2 34616.776} C_VEL
LIN {X 0,Y 753.102,Z 953.185,A -85,B 0,C 180,E1 34616.106,E2 34616.106} C_VEL
LIN {X 0,Y 753.194,Z 930.331,A -85,B 0,C 180,E1 34615.438,E2 34615.438} C_VEL
LIN {X 0,Y 753.279,Z 902.871,A -85,B 0,C 180,E1 34614.799,E2 34614.799} C_VEL
LIN {X 0,Y 753.353,Z 875.541,A -85,B 0,C 180,E1 34614.33,E2 34614.33} C_VEL
LIN {X 0,Y 753.602,Z 629.106,A -85,B 0,C 180,E1 34611.438,E2 34611.438} C_VEL
LIN {X 0,Y 753.802,Z 421.326,A -85,B 0,C 180,E1 34608.927,E2 34608.927} C_VEL
LIN {X 0,Y 753.643,Z 399.66,A -85,B 0,C 180,E1 34608.648,E2 34608.648} C_VEL
LIN {X 0,Y 753.206,Z 397.471,A -85,B 0,C 180,E1 34608.564,E2 34608.564} C_VEL
LIN {X 0,Y 753.076,Z 390.764,A -85,B 0,C 180,E1 34608.097,E2 34608.097} C_VEL
LIN {X 0,Y 751.966,Z 387.567,A -85,B 0,C 180,E1 34607.787,E2 34607.787} C_VEL
LIN {X 0,Y 751.95,Z 387.559,A -85,B 0,C 180,E1 34604.918,E2 34604.918} C_VEL
LIN {X 0,Y 751.96,Z 387.555,A -85,B 0,C 180,E1 34602.184,E2 34602.184} C_VEL
LIN {X 0,Y 751.975,Z 387.566,A -85,B 0,C 180,E1 34599.267,E2 34599.267} C_VEL
LIN {X 0,Y 751.971,Z 387.553,A -85,B 0,C 180,E1 34596.279,E2 34596.279} C_VEL
LIN {X 0,Y 751.959,Z 387.562,A -85,B 0,C 180,E1 34593.31,E2 34593.31} C_VEL
LIN {X 0,Y 751.952,Z 387.556,A -85,B 0,C 180,E1 34590.44,E2 34590.44} C_VEL
LIN {X 0,Y 751.955,Z 387.555,A -85,B 0,C 180,E1 34587.65,E2 34587.65} C_VEL
LIN {X 0,Y 751.97,Z 387.565,A -85,B 0,C 180,E1 34584.744,E2 34584.744} C_VEL
LIN {X 0,Y 751.971,Z 387.552,A -85,B 0,C 180,E1 34581.694,E2 34581.694} C_VEL
LIN {X 0,Y 751.963,Z 387.563,A -85,B 0,C 180,E1 34578.691,E2 34578.691} C_VEL
LIN {X 0,Y 751.963,Z 387.553,A -85,B 0,C 180,E1 34575.739,E2 34575.739} C_VEL
LIN {X 0,Y 751.944,Z 387.557,A -85,B 0,C 180,E1 34572.987,E2 34572.987} C_VEL
LIN {X 0,Y 751.971,Z 387.562,A -85,B 0,C 180,E1 34570.109,E2 34570.109} C_VEL
LIN {X 0,Y 751.964,Z 387.553,A -85,B 0,C 180,E1 34567.104,E2 34567.104} C_VEL
LIN {X 0,Y 751.955,Z 387.564,A -85,B 0,C 180,E1 34564.194,E2 34564.194} C_VEL
LIN {X 0,Y 751.963,Z 387.556,A -85,B 0,C 180,E1 34561.295,E2 34561.295} C_VEL
LIN {X 0,Y 751.942,Z 387.556,A -85,B 0,C 180,E1 34558.552,E2 34558.552} C_VEL
LIN {X 0,Y 751.971,Z 387.562,A -85,B 0,C 180,E1 34555.73,E2 34555.73} C_VEL
LIN {X 0,Y 751.968,Z 387.552,A -85,B 0,C 180,E1 34552.666,E2 34552.666} C_VEL
LIN {X 0,Y 751.942,Z 387.559,A -85,B 0,C 180,E1 34549.813,E2 34549.813} C_VEL
LIN {X 0,Y 751.963,Z 387.559,A -85,B 0,C 180,E1 34547.014,E2 34547.014} C_VEL
LIN {X 0,Y 751.946,Z 387.554,A -85,B 0,C 180,E1 34544.181,E2 34544.181} C_VEL
LIN {X 0,Y 751.949,Z 387.564,A -85,B 0,C 180,E1 34541.389,E2 34541.389} C_VEL
LIN {X 0,Y 751.969,Z 387.556,A -85,B 0,C 180,E1 34538.469,E2 34538.469} C_VEL
LIN {X 0,Y 751.935,Z 387.557,A -85,B 0,C 180,E1 34535.739,E2 34535.739} C_VEL
LIN {X 0,Y 751.958,Z 387.564,A -85,B 0,C 180,E1 34532.95,E2 34532.95} C_VEL
LIN {X 0,Y 751.969,Z 387.552,A -85,B 0,C 180,E1 34529.914,E2 34529.914} C_VEL
LIN {X 0,Y 751.928,Z 387.561,A -85,B 0,C 180,E1 34527.143,E2 34527.143} C_VEL
LIN {X 0,Y 751.974,Z 387.564,A -85,B 0,C 180,E1 34524.38,E2 34524.38} C_VEL
LIN {X 0,Y 751.942,Z 387.557,A -85,B 0,C 180,E1 34521.417,E2 34521.417} C_VEL
LIN {X 0,Y 751.931,Z 387.564,A -85,B 0,C 180,E1 34518.706,E2 34518.706} C_VEL
LIN {X 0,Y 751.969,Z 387.563,A -85,B 0,C 180,E1 34515.832,E2 34515.832} C_VEL
LIN {X 0,Y 751.989,Z 387.688,A -85,B 0,C 180,E1 34514.048,E2 34514.048} C_VEL
LIN {X 0,Y 753.412,Z 391.775,A -85,B 0,C 180,E1 34513.672,E2 34513.672} C_VEL
LIN {X 0,Y 753.396,Z 428.088,A -85,B 0,C 180,E1 34511.343,E2 34511.343} C_VEL
LIN {X 0,Y 753.838,Z 431.094,A -85,B 0,C 180,E1 34511.276,E2 34511.276} C_VEL
LIN {X 0,Y 753.618,Z 646.938,A -85,B 0,C 180,E1 34508.661,E2 34508.661} C_VEL
LIN {X 0,Y 753.406,Z 872.523,A -85,B 0,C 180,E1 34506.024,E2 34506.024} C_VEL
LIN {X 0,Y 753.355,Z 910.206,A -85,B 0,C 180,E1 34505.556,E2 34505.556} C_VEL
LIN {X 0,Y 753.268,Z 936.352,A -85,B 0,C 180,E1 34505.082,E2 34505.082} C_VEL
LIN {X 0,Y 753.179,Z 962.785,A -85,B 0,C 180,E1 34504.453,E2 34504.453} C_VEL
LIN {X 0,Y 753.085,Z 990.533,A -85,B 0,C 180,E1 34503.62,E2 34503.62} C_VEL
LIN {X 0,Y 752.951,Z 1016.069,A -85,B 0,C 180,E1 34502.687,E2 34502.687} C_VEL
LIN {X 0,Y 752.854,Z 1036.625,A -85,B 0,C 180,E1 34501.823,E2 34501.823} C_VEL
LIN {X 0,Y 752.753,Z 1055.463,A -85,B 0,C 180,E1 34500.936,E2 34500.936} C_VEL
LIN {X 0,Y 752.661,Z 1074.779,A -85,B 0,C 180,E1 34499.925,E2 34499.925} C_VEL
LIN {X 0,Y 752.554,Z 1097.201,A -85,B 0,C 180,E1 34498.621,E2 34498.621} C_VEL
LIN {X 0,Y 752.422,Z 1119.191,A -85,B 0,C 180,E1 34497.162,E2 34497.162} C_VEL
LIN {X 0,Y 752.333,Z 1136.796,A -85,B 0,C 180,E1 34495.872,E2 34495.872} C_VEL
LIN {X 0,Y 752.229,Z 1156.824,A -85,B 0,C 180,E1 34494.253,E2 34494.253} C_VEL
LIN {X 0,Y 752.166,Z 1174.943,A -85,B 0,C 180,E1 34492.595,E2 34492.595} C_VEL
LIN {X 0,Y 752.101,Z 1189.586,A -85,B 0,C 180,E1 34491.12,E2 34491.12} C_VEL
LIN {X 0,Y 752.053,Z 1205.604,A -85,B 0,C 180,E1 34489.335,E2 34489.335} C_VEL
LIN {X 0,Y 751.968,Z 1220.062,A -85,B 0,C 180,E1 34487.491,E2 34487.491} C_VEL
LIN {X 0,Y 751.948,Z 1230.728,A -85,B 0,C 180,E1 34485.971,E2 34485.971} C_VEL
LIN {X 0,Y 751.959,Z 1240.573,A -85,B 0,C 180,E1 34484.401,E2 34484.401} C_VEL
LIN {X 0,Y 751.936,Z 1249.274,A -85,B 0,C 180,E1 34482.833,E2 34482.833} C_VEL
LIN {X 0,Y 751.919,Z 1257.2,A -85,B 0,C 180,E1 34481.198,E2 34481.198} C_VEL
LIN {X 0,Y 751.871,Z 1265.469,A -85,B 0,C 180,E1 34479.186,E2 34479.186} C_VEL
LIN {X 0,Y 751.912,Z 1272.561,A -85,B 0,C 180,E1 34476.954,E2 34476.954} C_VEL
LIN {X 0,Y 751.913,Z 1277.331,A -85,B 0,C 180,E1 34474.885,E2 34474.885} C_VEL
LIN {X 0,Y 751.912,Z 1280.335,A -85,B 0,C 180,E1 34472.9,E2 34472.9} C_VEL
LIN {X 0,Y 751.872,Z 1281.714,A -85,B 0,C 180,E1 34470.994,E2 34470.994} C_VEL
LIN {X 0,Y 751.863,Z 1281.828,A -85,B 0,C 180,E1 34469.394,E2 34469.394} C_VEL
LIN {X 0,Y 751.91,Z 1280.949,A -85,B 0,C 180,E1 34467.794,E2 34467.794} C_VEL
LIN {X 0,Y 751.915,Z 1278.809,A -85,B 0,C 180,E1 34465.962,E2 34465.962} C_VEL
LIN {X 0,Y 751.916,Z 1274.743,A -85,B 0,C 180,E1 34463.897,E2 34463.897} C_VEL
LIN {X 0,Y 751.898,Z 1269.34,A -85,B 0,C 180,E1 34461.977,E2 34461.977} C_VEL
LIN {X 0,Y 751.905,Z 1263.025,A -85,B 0,C 180,E1 34460.195,E2 34460.195} C_VEL
LIN {X 0,Y 751.928,Z 1256.16,A -85,B 0,C 180,E1 34458.576,E2 34458.576} C_VEL
LIN {X 0,Y 751.919,Z 1248.491,A -85,B 0,C 180,E1 34457.017,E2 34457.017} C_VEL
LIN {X 0,Y 751.96,Z 1239.685,A -85,B 0,C 180,E1 34455.449,E2 34455.449} C_VEL
LIN {X 0,Y 751.959,Z 1228.627,A -85,B 0,C 180,E1 34453.71,E2 34453.71} C_VEL
LIN {X 0,Y 752.025,Z 1213.411,A -85,B 0,C 180,E1 34451.637,E2 34451.637} C_VEL
LIN {X 0,Y 752.039,Z 1200.252,A -85,B 0,C 180,E1 34450.054,E2 34450.054} C_VEL
LIN {X 0,Y 752.115,Z 1186.537,A -85,B 0,C 180,E1 34448.561,E2 34448.561} C_VEL
LIN {X 0,Y 752.193,Z 1168.553,A -85,B 0,C 180,E1 34446.793,E2 34446.793} C_VEL
LIN {X 0,Y 752.282,Z 1150.274,A -85,B 0,C 180,E1 34445.204,E2 34445.204} C_VEL
LIN {X 0,Y 752.333,Z 1132.797,A -85,B 0,C 180,E1 34443.822,E2 34443.822} C_VEL
LIN {X 0,Y 752.475,Z 1109.939,A -85,B 0,C 180,E1 34442.204,E2 34442.204} C_VEL
LIN {X 0,Y 752.577,Z 1090.085,A -85,B 0,C 180,E1 34440.955,E2 34440.955} C_VEL
LIN {X 0,Y 752.669,Z 1071.713,A -85,B 0,C 180,E1 34439.907,E2 34439.907} C_VEL
LIN {X 0,Y 752.768,Z 1051.175,A -85,B 0,C 180,E1 34438.85,E2 34438.85} C_VEL
LIN {X 0,Y 752.93,Z 1024.435,A -85,B 0,C 180,E1 34437.65,E2 34437.65} C_VEL
LIN {X 0,Y 753.025,Z 1003.541,A -85,B 0,C 180,E1 34436.84,E2 34436.84} C_VEL
LIN {X 0,Y 753.102,Z 983.478,A -85,B 0,C 180,E1 34436.16,E2 34436.16} C_VEL
LIN {X 0,Y 753.192,Z 960.56,A -85,B 0,C 180,E1 34435.489,E2 34435.489} C_VEL
LIN {X 0,Y 753.277,Z 933.06,A -85,B 0,C 180,E1 34434.848,E2 34434.848} C_VEL
LIN {X 0,Y 753.357,Z 906.078,A -85,B 0,C 180,E1 34434.383,E2 34434.383} C_VEL
LIN {X 0,Y 753.486,Z 778.403,A -85,B 0,C 180,E1 34432.886,E2 34432.886} C_VEL
LIN {X 0,Y 753.71,Z 556.709,A -85,B 0,C 180,E1 34430.258,E2 34430.258} C_VEL
LIN {X 0,Y 753.681,Z 429.212,A -85,B 0,C 180,E1 34428.69,E2 34428.69} C_VEL
LIN {X 0,Y 753.276,Z 427.36,A -85,B 0,C 180,E1 34428.628,E2 34428.628} C_VEL
LIN {X 0,Y 753.309,Z 391.095,A -85,B 0,C 180,E1 34426.275,E2 34426.275} C_VEL
LIN {X 0,Y 751.971,Z 387.567,A -85,B 0,C 180,E1 34425.92,E2 34425.92} C_VEL
LIN {X 0,Y 751.916,Z 387.563,A -85,B 0,C 180,E1 34423.223,E2 34423.223} C_VEL
LIN {X 0,Y 751.949,Z 387.555,A -85,B 0,C 180,E1 34420.56,E2 34420.56} C_VEL
LIN {X 0,Y 751.937,Z 387.565,A -85,B 0,C 180,E1 34417.519,E2 34417.519} C_VEL
LIN {X 0,Y 751.905,Z 387.562,A -85,B 0,C 180,E1 34414.97,E2 34414.97} C_VEL
LIN {X 0,Y 751.92,Z 387.56,A -85,B 0,C 180,E1 34412.496,E2 34412.496} C_VEL
LIN {X 0,Y 751.962,Z 387.565,A -85,B 0,C 180,E1 34409.559,E2 34409.559} C_VEL
LIN {X 0,Y 751.898,Z 387.564,A -85,B 0,C 180,E1 34406.967,E2 34406.967} C_VEL
LIN {X 0,Y 751.888,Z 387.562,A -85,B 0,C 180,E1 34404.598,E2 34404.598} C_VEL
LIN {X 0,Y 751.908,Z 387.563,A -85,B 0,C 180,E1 34402.189,E2 34402.189} C_VEL
LIN {X 0,Y 751.927,Z 387.566,A -85,B 0,C 180,E1 34399.175,E2 34399.175} C_VEL
LIN {X 0,Y 751.881,Z 387.565,A -85,B 0,C 180,E1 34396.693,E2 34396.693} C_VEL
LIN {X 0,Y 751.872,Z 387.563,A -85,B 0,C 180,E1 34394.478,E2 34394.478} C_VEL
LIN {X 0,Y 751.869,Z 387.566,A -85,B 0,C 180,E1 34392.285,E2 34392.285} C_VEL
LIN {X 0,Y 751.879,Z 387.565,A -85,B 0,C 180,E1 34389.955,E2 34389.955} C_VEL
LIN {X 0,Y 751.95,Z 387.567,A -85,B 0,C 180,E1 34387.104,E2 34387.104} C_VEL
LIN {X 0,Y 751.873,Z 387.564,A -85,B 0,C 180,E1 34384.424,E2 34384.424} C_VEL
LIN {X 0,Y 751.868,Z 387.564,A -85,B 0,C 180,E1 34382.21,E2 34382.21} C_VEL
LIN {X 0,Y 751.873,Z 387.565,A -85,B 0,C 180,E1 34380,E2 34380} C_VEL
LIN {X 0,Y 751.886,Z 387.564,A -85,B 0,C 180,E1 34377.714,E2 34377.714} C_VEL
LIN {X 0,Y 751.978,Z 387.565,A -85,B 0,C 180,E1 34374.965,E2 34374.965} C_VEL
LIN {X 0,Y 751.9,Z 387.563,A -85,B 0,C 180,E1 34374.298,E2 34374.298} C_VEL
LIN {X 0,Y 750.876,Z 387.694,A -85,B 0,C 180,E1 34373.711,E2 34373.711} C_VEL
LIN {X 0,Y 744.465,Z 388.488,A -85,B 0,C 180,E1 34372.066,E2 34372.066} C_VEL
LIN {X 0,Y 743.952,Z 388.551,A -85,B 0,C 180,E1 34371.639,E2 34371.639} C_VEL
LIN {X 0,Y 744.033,Z 388.554,A -85,B 0,C 180,E1 34368.92,E2 34368.92} C_VEL
LIN {X 0,Y 743.974,Z 388.547,A -85,B 0,C 180,E1 34366.08,E2 34366.08} C_VEL
LIN {X 0,Y 743.96,Z 388.55,A -85,B 0,C 180,E1 34363.606,E2 34363.606} C_VEL
LIN {X 0,Y 744,Z 388.554,A -85,B 0,C 180,E1 34361.02,E2 34361.02} C_VEL
LIN {X 0,Y 743.997,Z 388.547,A -85,B 0,C 180,E1 34357.978,E2 34357.978} C_VEL
LIN {X 0,Y 743.972,Z 388.55,A -85,B 0,C 180,E1 34355.377,E2 34355.377} C_VEL
LIN {X 0,Y 744.033,Z 388.554,A -85,B 0,C 180,E1 34352.638,E2 34352.638} C_VEL
LIN {X 0,Y 743.997,Z 388.542,A -85,B 0,C 180,E1 34349.647,E2 34349.647} C_VEL
LIN {X 0,Y 743.993,Z 388.553,A -85,B 0,C 180,E1 34346.931,E2 34346.931} C_VEL
LIN {X 0,Y 744.03,Z 388.55,A -85,B 0,C 180,E1 34344.121,E2 34344.121} C_VEL
LIN {X 0,Y 743.999,Z 388.543,A -85,B 0,C 180,E1 34341.323,E2 34341.323} C_VEL
LIN {X 0,Y 744.021,Z 388.555,A -85,B 0,C 180,E1 34338.506,E2 34338.506} C_VEL
LIN {X 0,Y 744.029,Z 388.546,A -85,B 0,C 180,E1 34335.411,E2 34335.411} C_VEL
LIN {X 0,Y 744.029,Z 388.708,A -85,B 0,C 180,E1 34332.585,E2 34332.585} C_VEL
LIN {X 0,Y 745.478,Z 392.24,A -85,B 0,C 180,E1 34332.236,E2 34332.236} C_VEL
LIN {X 0,Y 746.579,Z 395.552,A -85,B 0,C 180,E1 34331.929,E2 34331.929} C_VEL
LIN {X 0,Y 746.704,Z 398.595,A -85,B 0,C 180,E1 34331.745,E2 34331.745} C_VEL
LIN {X 0,Y 747.785,Z 403.281,A -85,B 0,C 180,E1 34331.612,E2 34331.612} C_VEL
LIN {X 0,Y 747.369,Z 612.825,A -85,B 0,C 180,E1 34329.05,E2 34329.05} C_VEL
LIN {X 0,Y 746.934,Z 837.895,A -85,B 0,C 180,E1 34326.395,E2 34326.395} C_VEL
LIN {X 0,Y 746.826,Z 879.405,A -85,B 0,C 180,E1 34325.882,E2 34325.882} C_VEL
LIN {X 0,Y 746.66,Z 905.728,A -85,B 0,C 180,E1 34325.408,E2 34325.408} C_VEL
LIN {X 0,Y 746.488,Z 932.26,A -85,B 0,C 180,E1 34324.774,E2 34324.774} C_VEL
LIN {X 0,Y 746.3,Z 957.922,A -85,B 0,C 180,E1 34324.005,E2 34324.005} C_VEL
LIN {X 0,Y 746.02,Z 984.397,A -85,B 0,C 180,E1 34323.053,E2 34323.053} C_VEL
LIN {X 0,Y 745.82,Z 1005.826,A -85,B 0,C 180,E1 34322.151,E2 34322.151} C_VEL
LIN {X 0,Y 745.617,Z 1025.716,A -85,B 0,C 180,E1 34321.208,E2 34321.208} C_VEL
LIN {X 0,Y 745.421,Z 1046.522,A -85,B 0,C 180,E1 34320.105,E2 34320.105} C_VEL
LIN {X 0,Y 745.125,Z 1071.312,A -85,B 0,C 180,E1 34318.618,E2 34318.618} C_VEL
LIN {X 0,Y 744.939,Z 1090.684,A -85,B 0,C 180,E1 34317.306,E2 34317.306} C_VEL
LIN {X 0,Y 744.767,Z 1108.858,A -85,B 0,C 180,E1 34315.95,E2 34315.95} C_VEL
LIN {X 0,Y 744.525,Z 1130.14,A -85,B 0,C 180,E1 34314.175,E2 34314.175} C_VEL
LIN {X 0,Y 744.429,Z 1145.415,A -85,B 0,C 180,E1 34312.752,E2 34312.752} C_VEL
LIN {X 0,Y 744.305,Z 1160.587,A -85,B 0,C 180,E1 34311.201,E2 34311.201} C_VEL
LIN {X 0,Y 744.177,Z 1177.9,A -85,B 0,C 180,E1 34309.215,E2 34309.215} C_VEL
LIN {X 0,Y 744.066,Z 1190.375,A -85,B 0,C 180,E1 34307.595,E2 34307.595} C_VEL
LIN {X 0,Y 744.012,Z 1200.948,A -85,B 0,C 180,E1 34306.067,E2 34306.067} C_VEL
LIN {X 0,Y 744.008,Z 1210.354,A -85,B 0,C 180,E1 34304.551,E2 34304.551} C_VEL
LIN {X 0,Y 743.947,Z 1219.079,A -85,B 0,C 180,E1 34302.966,E2 34302.966} C_VEL
LIN {X 0,Y 743.947,Z 1227.029,A -85,B 0,C 180,E1 34301.312,E2 34301.312} C_VEL
LIN {X 0,Y 743.881,Z 1235.328,A -85,B 0,C 180,E1 34299.278,E2 34299.278} C_VEL
LIN {X 0,Y 743.918,Z 1242.454,A -85,B 0,C 180,E1 34297.022,E2 34297.022} C_VEL
LIN {X 0,Y 743.916,Z 1247.11,A -85,B 0,C 180,E1 34295.008,E2 34295.008} C_VEL
LIN {X 0,Y 743.911,Z 1250.275,A -85,B 0,C 180,E1 34292.954,E2 34292.954} C_VEL
LIN {X 0,Y 743.877,Z 1251.703,A -85,B 0,C 180,E1 34290.998,E2 34290.998} C_VEL
LIN {X 0,Y 743.865,Z 1251.839,A -85,B 0,C 180,E1 34289.38,E2 34289.38} C_VEL
LIN {X 0,Y 743.907,Z 1250.982,A -85,B 0,C 180,E1 34287.763,E2 34287.763} C_VEL
LIN {X 0,Y 743.917,Z 1248.87,A -85,B 0,C 180,E1 34285.912,E2 34285.912} C_VEL
LIN {X 0,Y 743.921,Z 1244.649,A -85,B 0,C 180,E1 34283.747,E2 34283.747} C_VEL
LIN {X 0,Y 743.927,Z 1238.953,A -85,B 0,C 180,E1 34281.728,E2 34281.728} C_VEL
LIN {X 0,Y 743.93,Z 1232.902,A -85,B 0,C 180,E1 34280.012,E2 34280.012} C_VEL
LIN {X 0,Y 743.938,Z 1225.976,A -85,B 0,C 180,E1 34278.366,E2 34278.366} C_VEL
LIN {X 0,Y 743.936,Z 1218.278,A -85,B 0,C 180,E1 34276.789,E2 34276.789} C_VEL
LIN {X 0,Y 743.988,Z 1208.976,A -85,B 0,C 180,E1 34275.123,E2 34275.123} C_VEL
LIN {X 0,Y 744.082,Z 1196.205,A -85,B 0,C 180,E1 34273.124,E2 34273.124} C_VEL
LIN {X 0,Y 744.159,Z 1182.422,A -85,B 0,C 180,E1 34271.266,E2 34271.266} C_VEL
LIN {X 0,Y 744.22,Z 1169.342,A -85,B 0,C 180,E1 34269.685,E2 34269.685} C_VEL
LIN {X 0,Y 744.327,Z 1154.551,A -85,B 0,C 180,E1 34268.069,E2 34268.069} C_VEL
LIN {X 0,Y 744.525,Z 1135.243,A -85,B 0,C 180,E1 34266.196,E2 34266.196} C_VEL
LIN {X 0,Y 744.655,Z 1118.873,A -85,B 0,C 180,E1 34264.771,E2 34264.771} C_VEL
LIN {X 0,Y 744.887,Z 1098.842,A -85,B 0,C 180,E1 34263.188,E2 34263.188} C_VEL
LIN {X 0,Y 745.073,Z 1077.312,A -85,B 0,C 180,E1 34261.686,E2 34261.686} C_VEL
LIN {X 0,Y 745.274,Z 1058.489,A -85,B 0,C 180,E1 34260.501,E2 34260.501} C_VEL
LIN {X 0,Y 745.486,Z 1037.166,A -85,B 0,C 180,E1 34259.289,E2 34259.289} C_VEL
LIN {X 0,Y 745.785,Z 1011.591,A -85,B 0,C 180,E1 34258.021,E2 34258.021} C_VEL
LIN {X 0,Y 745.986,Z 990.863,A -85,B 0,C 180,E1 34257.12,E2 34257.12} C_VEL
LIN {X 0,Y 746.17,Z 970.738,A -85,B 0,C 180,E1 34256.349,E2 34256.349} C_VEL
LIN {X 0,Y 746.336,Z 950.97,A -85,B 0,C 180,E1 34255.687,E2 34255.687} C_VEL
LIN {X 0,Y 746.517,Z 928.701,A -85,B 0,C 180,E1 34255.042,E2 34255.042} C_VEL
LIN {X 0,Y 746.703,Z 901.863,A -85,B 0,C 180,E1 34254.422,E2 34254.422} C_VEL
LIN {X 0,Y 746.835,Z 873.754,A -85,B 0,C 180,E1 34253.945,E2 34253.945} C_VEL
LIN {X 0,Y 747.323,Z 633.001,A -85,B 0,C 180,E1 34251.101,E2 34251.101} C_VEL
LIN {X 0,Y 747.745,Z 425.588,A -85,B 0,C 180,E1 34248.576,E2 34248.576} C_VEL
LIN {X 0,Y 747.627,Z 401.847,A -85,B 0,C 180,E1 34248.269,E2 34248.269} C_VEL
LIN {X 0,Y 746.559,Z 397.737,A -85,B 0,C 180,E1 34248.131,E2 34248.131} C_VEL
LIN {X 0,Y 746.4,Z 394.778,A -85,B 0,C 180,E1 34247.915,E2 34247.915} C_VEL
LIN {X 0,Y 744.014,Z 388.555,A -85,B 0,C 180,E1 34247.287,E2 34247.287} C_VEL
LIN {X 0,Y 744.03,Z 388.545,A -85,B 0,C 180,E1 34244.36,E2 34244.36} C_VEL
LIN {X 0,Y 744.035,Z 388.556,A -85,B 0,C 180,E1 34241.391,E2 34241.391} C_VEL
LIN {X 0,Y 744.027,Z 388.544,A -85,B 0,C 180,E1 34238.38,E2 34238.38} C_VEL
LIN {X 0,Y 744.017,Z 388.552,A -85,B 0,C 180,E1 34235.47,E2 34235.47} C_VEL
LIN {X 0,Y 744.015,Z 388.55,A -85,B 0,C 180,E1 34232.701,E2 34232.701} C_VEL
LIN {X 0,Y 744.024,Z 388.539,A -85,B 0,C 180,E1 34229.818,E2 34229.818} C_VEL
LIN {X 0,Y 744.039,Z 388.552,A -85,B 0,C 180,E1 34226.832,E2 34226.832} C_VEL
LIN {X 0,Y 744.036,Z 388.541,A -85,B 0,C 180,E1 34223.768,E2 34223.768} C_VEL
LIN {X 0,Y 744.024,Z 388.552,A -85,B 0,C 180,E1 34220.781,E2 34220.781} C_VEL
LIN {X 0,Y 744.022,Z 388.545,A -85,B 0,C 180,E1 34217.843,E2 34217.843} C_VEL
LIN {X 0,Y 744.005,Z 388.544,A -85,B 0,C 180,E1 34215.033,E2 34215.033} C_VEL
LIN {X 0,Y 744.031,Z 388.554,A -85,B 0,C 180,E1 34212.18,E2 34212.18} C_VEL
LIN {X 0,Y 744.028,Z 388.537,A -85,B 0,C 180,E1 34209.202,E2 34209.202} C_VEL
LIN {X 0,Y 744.02,Z 388.552,A -85,B 0,C 180,E1 34206.249,E2 34206.249} C_VEL
LIN {X 0,Y 744.027,Z 388.539,A -85,B 0,C 180,E1 34203.313,E2 34203.313} C_VEL
LIN {X 0,Y 744.001,Z 388.546,A -85,B 0,C 180,E1 34200.539,E2 34200.539} C_VEL
LIN {X 0,Y 744.034,Z 388.549,A -85,B 0,C 180,E1 34197.689,E2 34197.689} C_VEL
LIN {X 0,Y 744.023,Z 388.542,A -85,B 0,C 180,E1 34194.679,E2 34194.679} C_VEL
LIN {X 0,Y 744.009,Z 388.551,A -85,B 0,C 180,E1 34191.81,E2 34191.81} C_VEL
LIN {X 0,Y 744.025,Z 388.546,A -85,B 0,C 180,E1 34188.92,E2 34188.92} C_VEL
LIN {X 0,Y 744.002,Z 388.544,A -85,B 0,C 180,E1 34186.159,E2 34186.159} C_VEL
LIN {X 0,Y 744.027,Z 388.552,A -85,B 0,C 180,E1 34183.286,E2 34183.286} C_VEL
LIN {X 0,Y 744.02,Z 388.539,A -85,B 0,C 180,E1 34180.176,E2 34180.176} C_VEL
LIN {X 0,Y 743.998,Z 388.551,A -85,B 0,C 180,E1 34177.395,E2 34177.395} C_VEL
LIN {X 0,Y 744.028,Z 388.548,A -85,B 0,C 180,E1 34174.569,E2 34174.569} C_VEL
LIN {X 0,Y 744.006,Z 388.545,A -85,B 0,C 180,E1 34171.767,E2 34171.767} C_VEL
LIN {X 0,Y 744,Z 388.55,A -85,B 0,C 180,E1 34169.021,E2 34169.021} C_VEL
LIN {X 0,Y 744.029,Z 388.545,A -85,B 0,C 180,E1 34166.102,E2 34166.102} C_VEL
LIN {X 0,Y 743.994,Z 388.546,A -85,B 0,C 180,E1 34163.355,E2 34163.355} C_VEL
LIN {X 0,Y 744.007,Z 388.554,A -85,B 0,C 180,E1 34160.604,E2 34160.604} C_VEL
LIN {X 0,Y 744.036,Z 388.547,A -85,B 0,C 180,E1 34157.659,E2 34157.659} C_VEL
LIN {X 0,Y 743.985,Z 388.554,A -85,B 0,C 180,E1 34154.878,E2 34154.878} C_VEL
LIN {X 0,Y 744.006,Z 388.669,A -85,B 0,C 180,E1 34154.579,E2 34154.579} C_VEL
LIN {X 0,Y 745.358,Z 392.088,A -85,B 0,C 180,E1 34154.245,E2 34154.245} C_VEL
LIN {X 0,Y 746.911,Z 395.845,A -85,B 0,C 180,E1 34153.877,E2 34153.877} C_VEL
LIN {X 0,Y 746.793,Z 428.081,A -85,B 0,C 180,E1 34151.79,E2 34151.79} C_VEL
LIN {X 0,Y 747.807,Z 432.804,A -85,B 0,C 180,E1 34151.661,E2 34151.661} C_VEL
LIN {X 0,Y 747.357,Z 647.956,A -85,B 0,C 180,E1 34149.034,E2 34149.034} C_VEL
LIN {X 0,Y 746.924,Z 873.541,A -85,B 0,C 180,E1 34146.374,E2 34146.374} C_VEL
LIN {X 0,Y 746.821,Z 910.848,A -85,B 0,C 180,E1 34145.905,E2 34145.905} C_VEL
LIN {X 0,Y 746.655,Z 937.264,A -85,B 0,C 180,E1 34145.42,E2 34145.42} C_VEL
LIN {X 0,Y 746.477,Z 963.501,A -85,B 0,C 180,E1 34144.786,E2 34144.786} C_VEL
LIN {X 0,Y 746.257,Z 991.844,A -85,B 0,C 180,E1 34143.924,E2 34143.924} C_VEL
LIN {X 0,Y 746.007,Z 1016.408,A -85,B 0,C 180,E1 34143.016,E2 34143.016} C_VEL
LIN {X 0,Y 745.814,Z 1036.629,A -85,B 0,C 180,E1 34142.159,E2 34142.159} C_VEL
LIN {X 0,Y 745.615,Z 1056.357,A -85,B 0,C 180,E1 34141.221,E2 34141.221} C_VEL
LIN {X 0,Y 745.414,Z 1077.53,A -85,B 0,C 180,E1 34140.094,E2 34140.094} C_VEL
LIN {X 0,Y 745.121,Z 1101.873,A -85,B 0,C 180,E1 34138.626,E2 34138.626} C_VEL
LIN {X 0,Y 744.94,Z 1120.401,A -85,B 0,C 180,E1 34137.371,E2 34137.371} C_VEL
LIN {X 0,Y 744.767,Z 1138.232,A -85,B 0,C 180,E1 34136.043,E2 34136.043} C_VEL
LIN {X 0,Y 744.53,Z 1159.62,A -85,B 0,C 180,E1 34134.267,E2 34134.267} C_VEL
LIN {X 0,Y 744.425,Z 1175.798,A -85,B 0,C 180,E1 34132.76,E2 34132.76} C_VEL
LIN {X 0,Y 744.299,Z 1191.927,A -85,B 0,C 180,E1 34131.105,E2 34131.105} C_VEL
LIN {X 0,Y 744.167,Z 1208.841,A -85,B 0,C 180,E1 34129.141,E2 34129.141} C_VEL
LIN {X 0,Y 744.064,Z 1220.646,A -85,B 0,C 180,E1 34127.602,E2 34127.602} C_VEL
LIN {X 0,Y 744.015,Z 1231.193,A -85,B 0,C 180,E1 34126.075,E2 34126.075} C_VEL
LIN {X 0,Y 744.005,Z 1241.04,A -85,B 0,C 180,E1 34124.479,E2 34124.479} C_VEL
LIN {X 0,Y 743.971,Z 1250.507,A -85,B 0,C 180,E1 34122.736,E2 34122.736} C_VEL
LIN {X 0,Y 743.926,Z 1260.583,A -85,B 0,C 180,E1 34120.535,E2 34120.535} C_VEL
LIN {X 0,Y 743.906,Z 1267.268,A -85,B 0,C 180,E1 34118.739,E2 34118.739} C_VEL
LIN {X 0,Y 743.912,Z 1272.971,A -85,B 0,C 180,E1 34116.874,E2 34116.874} C_VEL
LIN {X 0,Y 743.909,Z 1277.627,A -85,B 0,C 180,E1 34114.783,E2 34114.783} C_VEL
LIN {X 0,Y 743.915,Z 1280.403,A -85,B 0,C 180,E1 34112.854,E2 34112.854} C_VEL
LIN {X 0,Y 743.873,Z 1281.714,A -85,B 0,C 180,E1 34111.005,E2 34111.005} C_VEL
LIN {X 0,Y 743.863,Z 1281.828,A -85,B 0,C 180,E1 34109.387,E2 34109.387} C_VEL
LIN {X 0,Y 743.909,Z 1280.949,A -85,B 0,C 180,E1 34107.77,E2 34107.77} C_VEL
LIN {X 0,Y 743.916,Z 1278.809,A -85,B 0,C 180,E1 34105.919,E2 34105.919} C_VEL
LIN {X 0,Y 743.92,Z 1274.743,A -85,B 0,C 180,E1 34103.831,E2 34103.831} C_VEL
LIN {X 0,Y 743.91,Z 1269.341,A -85,B 0,C 180,E1 34101.891,E2 34101.891} C_VEL
LIN {X 0,Y 743.926,Z 1263.059,A -85,B 0,C 180,E1 34100.098,E2 34100.098} C_VEL
LIN {X 0,Y 743.94,Z 1256.161,A -85,B 0,C 180,E1 34098.452,E2 34098.452} C_VEL
LIN {X 0,Y 743.939,Z 1248.492,A -85,B 0,C 180,E1 34096.875,E2 34096.875} C_VEL
LIN {X 0,Y 743.997,Z 1239.687,A -85,B 0,C 180,E1 34095.29,E2 34095.29} C_VEL
LIN {X 0,Y 744.042,Z 1228.629,A -85,B 0,C 180,E1 34093.532,E2 34093.532} C_VEL
LIN {X 0,Y 744.15,Z 1213.414,A -85,B 0,C 180,E1 34091.436,E2 34091.436} C_VEL
LIN {X 0,Y 744.205,Z 1200.71,A -85,B 0,C 180,E1 34089.887,E2 34089.887} C_VEL
LIN {X 0,Y 744.327,Z 1186.986,A -85,B 0,C 180,E1 34088.373,E2 34088.373} C_VEL
LIN {X 0,Y 744.48,Z 1169.901,A -85,B 0,C 180,E1 34086.664,E2 34086.664} C_VEL
LIN {X 0,Y 744.655,Z 1150.877,A -85,B 0,C 180,E1 34084.983,E2 34084.983} C_VEL
LIN {X 0,Y 744.781,Z 1133.904,A -85,B 0,C 180,E1 34083.622,E2 34083.622} C_VEL
LIN {X 0,Y 745.052,Z 1112.59,A -85,B 0,C 180,E1 34082.077,E2 34082.077} C_VEL
LIN {X 0,Y 745.261,Z 1090.789,A -85,B 0,C 180,E1 34080.685,E2 34080.685} C_VEL
LIN {X 0,Y 745.441,Z 1071.936,A -85,B 0,C 180,E1 34079.597,E2 34079.597} C_VEL
LIN {X 0,Y 745.651,Z 1051.267,A -85,B 0,C 180,E1 34078.524,E2 34078.524} C_VEL
LIN {X 0,Y 745.968,Z 1024.439,A -85,B 0,C 180,E1 34077.311,E2 34077.311} C_VEL
LIN {X 0,Y 746.162,Z 1002.602,A -85,B 0,C 180,E1 34076.461,E2 34076.461} C_VEL
LIN {X 0,Y 746.326,Z 982.749,A -85,B 0,C 180,E1 34075.787,E2 34075.787} C_VEL
LIN {X 0,Y 746.509,Z 960.136,A -85,B 0,C 180,E1 34075.124,E2 34075.124} C_VEL
LIN {X 0,Y 746.686,Z 932.999,A -85,B 0,C 180,E1 34074.49,E2 34074.49} C_VEL
LIN {X 0,Y 746.83,Z 905.682,A -85,B 0,C 180,E1 34074.018,E2 34074.018} C_VEL
LIN {X 0,Y 747.327,Z 661.55,A -85,B 0,C 180,E1 34071.129,E2 34071.129} C_VEL
LIN {X 0,Y 747.759,Z 452.109,A -85,B 0,C 180,E1 34068.578,E2 34068.578} C_VEL
LIN {X 0,Y 747.624,Z 431.169,A -85,B 0,C 180,E1 34068.306,E2 34068.306} C_VEL
LIN {X 0,Y 746.678,Z 427.36,A -85,B 0,C 180,E1 34068.181,E2 34068.181} C_VEL
LIN {X 0,Y 746.8,Z 395.358,A -85,B 0,C 180,E1 34066.082,E2 34066.082} C_VEL
LIN {X 0,Y 745.356,Z 392.092,A -85,B 0,C 180,E1 34065.755,E2 34065.755} C_VEL
LIN {X 0,Y 743.985,Z 388.557,A -85,B 0,C 180,E1 34065.386,E2 34065.386} C_VEL
LIN {X 0,Y 744.004,Z 388.55,A -85,B 0,C 180,E1 34062.691,E2 34062.691} C_VEL
LIN {X 0,Y 744.012,Z 388.556,A -85,B 0,C 180,E1 34059.65,E2 34059.65} C_VEL
LIN {X 0,Y 743.968,Z 388.55,A -85,B 0,C 180,E1 34057.021,E2 34057.021} C_VEL
LIN {X 0,Y 744,Z 388.547,A -85,B 0,C 180,E1 34054.405,E2 34054.405} C_VEL
LIN {X 0,Y 743.988,Z 388.553,A -85,B 0,C 180,E1 34051.34,E2 34051.34} C_VEL
LIN {X 0,Y 743.957,Z 388.551,A -85,B 0,C 180,E1 34048.815,E2 34048.815} C_VEL
LIN {X 0,Y 743.973,Z 388.55,A -85,B 0,C 180,E1 34046.321,E2 34046.321} C_VEL
LIN {X 0,Y 744.008,Z 388.555,A -85,B 0,C 180,E1 34043.357,E2 34043.357} C_VEL
LIN {X 0,Y 743.949,Z 388.55,A -85,B 0,C 180,E1 34040.783,E2 34040.783} C_VEL
LIN {X 0,Y 743.94,Z 388.553,A -85,B 0,C 180,E1 34038.493,E2 34038.493} C_VEL
LIN {X 0,Y 743.948,Z 388.553,A -85,B 0,C 180,E1 34036.154,E2 34036.154} C_VEL
LIN {X 0,Y 744.025,Z 388.556,A -85,B 0,C 180,E1 34033.286,E2 34033.286} C_VEL
LIN {X 0,Y 743.936,Z 388.554,A -85,B 0,C 180,E1 34030.611,E2 34030.611} C_VEL
LIN {X 0,Y 743.924,Z 388.553,A -85,B 0,C 180,E1 34028.347,E2 34028.347} C_VEL
LIN {X 0,Y 743.923,Z 388.556,A -85,B 0,C 180,E1 34026.173,E2 34026.173} C_VEL
LIN {X 0,Y 743.938,Z 388.553,A -85,B 0,C 180,E1 34023.853,E2 34023.853} C_VEL
LIN {X 0,Y 744.032,Z 388.554,A -85,B 0,C 180,E1 34021.001,E2 34021.001} C_VEL
LIN {X 0,Y 743.947,Z 388.551,A -85,B 0,C 180,E1 34018.306,E2 34018.306} C_VEL
LIN {X 0,Y 743.941,Z 388.551,A -85,B 0,C 180,E1 34015.992,E2 34015.992} C_VEL
LIN {X 0,Y 743.951,Z 388.554,A -85,B 0,C 180,E1 34013.673,E2 34013.673} C_VEL
LIN {X 0,Y 743.952,Z 388.551,A -85,B 0,C 180,E1 34011.639,E2 34011.639} C_VEL
LIN {X 0,Y 742.98,Z 388.681,A -85,B 0,C 180,E1 34011.046,E2 34011.046} C_VEL
LIN {X 0,Y 736.583,Z 389.472,A -85,B 0,C 180,E1 34009.385,E2 34009.385} C_VEL
LIN {X 0,Y 736.089,Z 389.542,A -85,B 0,C 180,E1 34008.953,E2 34008.953} C_VEL
LIN {X 0,Y 736.036,Z 389.535,A -85,B 0,C 180,E1 34006.087,E2 34006.087} C_VEL
LIN {X 0,Y 736.022,Z 389.539,A -85,B 0,C 180,E1 34003.586,E2 34003.586} C_VEL
LIN {X 0,Y 736.069,Z 389.544,A -85,B 0,C 180,E1 34000.969,E2 34000.969} C_VEL
LIN {X 0,Y 736.059,Z 389.536,A -85,B 0,C 180,E1 33997.98,E2 33997.98} C_VEL
LIN {X 0,Y 736.035,Z 389.539,A -85,B 0,C 180,E1 33995.327,E2 33995.327} C_VEL
LIN {X 0,Y 736.097,Z 389.543,A -85,B 0,C 180,E1 33992.581,E2 33992.581} C_VEL
LIN {X 0,Y 736.055,Z 389.53,A -85,B 0,C 180,E1 33989.598,E2 33989.598} C_VEL
LIN {X 0,Y 736.056,Z 389.542,A -85,B 0,C 180,E1 33986.9,E2 33986.9} C_VEL
LIN {X 0,Y 736.094,Z 389.536,A -85,B 0,C 180,E1 33983.972,E2 33983.972} C_VEL
LIN {X 0,Y 736.053,Z 389.533,A -85,B 0,C 180,E1 33981.126,E2 33981.126} C_VEL
LIN {X 0,Y 736.099,Z 389.544,A -85,B 0,C 180,E1 33978.331,E2 33978.331} C_VEL
LIN {X 0,Y 736.077,Z 389.537,A -85,B 0,C 180,E1 33975.279,E2 33975.279} C_VEL
LIN {X 0,Y 736.079,Z 389.616,A -85,B 0,C 180,E1 33973.092,E2 33973.092} C_VEL
LIN {X 0,Y 737.164,Z 392.708,A -85,B 0,C 180,E1 33972.793,E2 33972.793} C_VEL
LIN {X 0,Y 739.791,Z 398.545,A -85,B 0,C 180,E1 33972.226,E2 33972.226} C_VEL
LIN {X 0,Y 741.249,Z 402.765,A -85,B 0,C 180,E1 33972.069,E2 33972.069} C_VEL
LIN {X 0,Y 741.785,Z 405.624,A -85,B 0,C 180,E1 33971.995,E2 33971.995} C_VEL
LIN {X 0,Y 741.144,Z 614.275,A -85,B 0,C 180,E1 33969.424,E2 33969.424} C_VEL
LIN {X 0,Y 740.484,Z 839.727,A -85,B 0,C 180,E1 33966.743,E2 33966.743} C_VEL
LIN {X 0,Y 740.321,Z 880.04,A -85,B 0,C 180,E1 33966.238,E2 33966.238} C_VEL
LIN {X 0,Y 740.076,Z 906.654,A -85,B 0,C 180,E1 33965.751,E2 33965.751} C_VEL
LIN {X 0,Y 739.818,Z 932.917,A -85,B 0,C 180,E1 33965.116,E2 33965.116} C_VEL
LIN {X 0,Y 739.525,Z 959.893,A -85,B 0,C 180,E1 33964.298,E2 33964.298} C_VEL
LIN {X 0,Y 739.103,Z 985.533,A -85,B 0,C 180,E1 33963.356,E2 33963.356} C_VEL
LIN {X 0,Y 738.798,Z 1006.835,A -85,B 0,C 180,E1 33962.448,E2 33962.448} C_VEL
LIN {X 0,Y 738.492,Z 1027.355,A -85,B 0,C 180,E1 33961.46,E2 33961.46} C_VEL
LIN {X 0,Y 738.151,Z 1051.305,A -85,B 0,C 180,E1 33960.163,E2 33960.163} C_VEL
LIN {X 0,Y 737.73,Z 1073.971,A -85,B 0,C 180,E1 33958.755,E2 33958.755} C_VEL
LIN {X 0,Y 737.463,Z 1092.31,A -85,B 0,C 180,E1 33957.489,E2 33957.489} C_VEL
LIN {X 0,Y 737.18,Z 1113.238,A -85,B 0,C 180,E1 33955.891,E2 33955.891} C_VEL
LIN {X 0,Y 736.845,Z 1132.01,A -85,B 0,C 180,E1 33954.273,E2 33954.273} C_VEL
LIN {X 0,Y 736.687,Z 1147.129,A -85,B 0,C 180,E1 33952.836,E2 33952.836} C_VEL
LIN {X 0,Y 736.492,Z 1164.644,A -85,B 0,C 180,E1 33950.998,E2 33950.998} C_VEL
LIN {X 0,Y 736.295,Z 1179.84,A -85,B 0,C 180,E1 33949.181,E2 33949.181} C_VEL
LIN {X 0,Y 736.159,Z 1191.545,A -85,B 0,C 180,E1 33947.626,E2 33947.626} C_VEL
LIN {X 0,Y 736.079,Z 1201.998,A -85,B 0,C 180,E1 33946.083,E2 33946.083} C_VEL
LIN {X 0,Y 736.049,Z 1211.755,A -85,B 0,C 180,E1 33944.47,E2 33944.47} C_VEL
LIN {X 0,Y 735.994,Z 1222.357,A -85,B 0,C 180,E1 33942.47,E2 33942.47} C_VEL
LIN {X 0,Y 735.948,Z 1231.492,A -85,B 0,C 180,E1 33940.371,E2 33940.371} C_VEL
LIN {X 0,Y 735.916,Z 1237.658,A -85,B 0,C 180,E1 33938.67,E2 33938.67} C_VEL
LIN {X 0,Y 735.912,Z 1243.268,A -85,B 0,C 180,E1 33936.785,E2 33936.785} C_VEL
LIN {X 0,Y 735.906,Z 1247.852,A -85,B 0,C 180,E1 33934.672,E2 33934.672} C_VEL
LIN {X 0,Y 735.909,Z 1250.572,A -85,B 0,C 180,E1 33932.644,E2 33932.644} C_VEL
LIN {X 0,Y 735.873,Z 1251.725,A -85,B 0,C 180,E1 33930.931,E2 33930.931} C_VEL
LIN {X 0,Y 735.863,Z 1251.816,A -85,B 0,C 180,E1 33929.296,E2 33929.296} C_VEL
LIN {X 0,Y 735.904,Z 1250.914,A -85,B 0,C 180,E1 33927.66,E2 33927.66} C_VEL
LIN {X 0,Y 735.92,Z 1248.728,A -85,B 0,C 180,E1 33925.778,E2 33925.778} C_VEL
LIN {X 0,Y 735.923,Z 1244.647,A -85,B 0,C 180,E1 33923.678,E2 33923.678} C_VEL
LIN {X 0,Y 735.934,Z 1238.952,A -85,B 0,C 180,E1 33921.638,E2 33921.638} C_VEL
LIN {X 0,Y 735.945,Z 1232.901,A -85,B 0,C 180,E1 33919.903,E2 33919.903} C_VEL
LIN {X 0,Y 735.952,Z 1225.975,A -85,B 0,C 180,E1 33918.238,E2 33918.238} C_VEL
LIN {X 0,Y 735.962,Z 1218.276,A -85,B 0,C 180,E1 33916.643,E2 33916.643} C_VEL
LIN {X 0,Y 736.036,Z 1209.16,A -85,B 0,C 180,E1 33914.991,E2 33914.991} C_VEL
LIN {X 0,Y 736.16,Z 1196.771,A -85,B 0,C 180,E1 33913.018,E2 33913.018} C_VEL
LIN {X 0,Y 736.283,Z 1183.065,A -85,B 0,C 180,E1 33911.14,E2 33911.14} C_VEL
LIN {X 0,Y 736.394,Z 1170.009,A -85,B 0,C 180,E1 33909.537,E2 33909.537} C_VEL
LIN {X 0,Y 736.541,Z 1156.108,A -85,B 0,C 180,E1 33907.993,E2 33907.993} C_VEL
LIN {X 0,Y 736.826,Z 1137.566,A -85,B 0,C 180,E1 33906.145,E2 33906.145} C_VEL
LIN {X 0,Y 737.037,Z 1119.781,A -85,B 0,C 180,E1 33904.569,E2 33904.569} C_VEL
LIN {X 0,Y 737.302,Z 1102.161,A -85,B 0,C 180,E1 33903.152,E2 33903.152} C_VEL
LIN {X 0,Y 737.672,Z 1079.172,A -85,B 0,C 180,E1 33901.5,E2 33901.5} C_VEL
LIN {X 0,Y 737.968,Z 1059.938,A -85,B 0,C 180,E1 33900.269,E2 33900.269} C_VEL
LIN {X 0,Y 738.261,Z 1039.965,A -85,B 0,C 180,E1 33899.113,E2 33899.113} C_VEL
LIN {X 0,Y 738.725,Z 1015.557,A -85,B 0,C 180,E1 33897.861,E2 33897.861} C_VEL
LIN {X 0,Y 739.049,Z 991.97,A -85,B 0,C 180,E1 33896.818,E2 33896.818} C_VEL
LIN {X 0,Y 739.333,Z 970.847,A -85,B 0,C 180,E1 33896,E2 33896} C_VEL
LIN {X 0,Y 739.592,Z 950.221,A -85,B 0,C 180,E1 33895.306,E2 33895.306} C_VEL
LIN {X 0,Y 739.871,Z 927.316,A -85,B 0,C 180,E1 33894.646,E2 33894.646} C_VEL
LIN {X 0,Y 740.15,Z 900.887,A -85,B 0,C 180,E1 33894.04,E2 33894.04} C_VEL
LIN {X 0,Y 740.342,Z 873.541,A -85,B 0,C 180,E1 33893.576,E2 33893.576} C_VEL
LIN {X 0,Y 741.071,Z 636.801,A -85,B 0,C 180,E1 33890.757,E2 33890.757} C_VEL
LIN {X 0,Y 741.717,Z 429.578,A -85,B 0,C 180,E1 33888.215,E2 33888.215} C_VEL
LIN {X 0,Y 741.628,Z 404.076,A -85,B 0,C 180,E1 33887.884,E2 33887.884} C_VEL
LIN {X 0,Y 739.939,Z 398.826,A -85,B 0,C 180,E1 33887.698,E2 33887.698} C_VEL
LIN {X 0,Y 739.128,Z 396.941,A -85,B 0,C 180,E1 33887.557,E2 33887.557} C_VEL
LIN {X 0,Y 736.122,Z 389.852,A -85,B 0,C 180,E1 33886.838,E2 33886.838} C_VEL
LIN {X 0,Y 736.084,Z 389.54,A -85,B 0,C 180,E1 33886.727,E2 33886.727} C_VEL
LIN {X 0,Y 736.077,Z 389.543,A -85,B 0,C 180,E1 33883.836,E2 33883.836} C_VEL
LIN {X 0,Y 736.075,Z 389.541,A -85,B 0,C 180,E1 33881.004,E2 33881.004} C_VEL
LIN {X 0,Y 736.085,Z 389.534,A -85,B 0,C 180,E1 33878.076,E2 33878.076} C_VEL
LIN {X 0,Y 736.093,Z 389.537,A -85,B 0,C 180,E1 33875.071,E2 33875.071} C_VEL
LIN {X 0,Y 736.093,Z 389.531,A -85,B 0,C 180,E1 33872.044,E2 33872.044} C_VEL
LIN {X 0,Y 736.095,Z 389.539,A -85,B 0,C 180,E1 33868.979,E2 33868.979} C_VEL
LIN {X 0,Y 736.093,Z 389.526,A -85,B 0,C 180,E1 33865.938,E2 33865.938} C_VEL
LIN {X 0,Y 736.074,Z 389.54,A -85,B 0,C 180,E1 33863.031,E2 33863.031} C_VEL
LIN {X 0,Y 736.078,Z 389.534,A -85,B 0,C 180,E1 33860.172,E2 33860.172} C_VEL
LIN {X 0,Y 736.077,Z 389.534,A -85,B 0,C 180,E1 33857.307,E2 33857.307} C_VEL
LIN {X 0,Y 736.095,Z 389.536,A -85,B 0,C 180,E1 33854.394,E2 33854.394} C_VEL
LIN {X 0,Y 736.09,Z 389.531,A -85,B 0,C 180,E1 33851.28,E2 33851.28} C_VEL
LIN {X 0,Y 736.085,Z 389.535,A -85,B 0,C 180,E1 33848.279,E2 33848.279} C_VEL
LIN {X 0,Y 736.095,Z 389.531,A -85,B 0,C 180,E1 33845.222,E2 33845.222} C_VEL
LIN {X 0,Y 736.065,Z 389.532,A -85,B 0,C 180,E1 33842.336,E2 33842.336} C_VEL
LIN {X 0,Y 736.086,Z 389.539,A -85,B 0,C 180,E1 33839.533,E2 33839.533} C_VEL
LIN {X 0,Y 736.075,Z 389.525,A -85,B 0,C 180,E1 33836.651,E2 33836.651} C_VEL
LIN {X 0,Y 736.082,Z 389.542,A -85,B 0,C 180,E1 33833.761,E2 33833.761} C_VEL
LIN {X 0,Y 736.095,Z 389.525,A -85,B 0,C 180,E1 33830.698,E2 33830.698} C_VEL
LIN {X 0,Y 736.06,Z 389.539,A -85,B 0,C 180,E1 33827.845,E2 33827.845} C_VEL
LIN {X 0,Y 736.089,Z 389.537,A -85,B 0,C 180,E1 33825.043,E2 33825.043} C_VEL
LIN {X 0,Y 736.07,Z 389.534,A -85,B 0,C 180,E1 33822.121,E2 33822.121} C_VEL
LIN {X 0,Y 736.078,Z 389.537,A -85,B 0,C 180,E1 33819.234,E2 33819.234} C_VEL
LIN {X 0,Y 736.096,Z 389.53,A -85,B 0,C 180,E1 33816.207,E2 33816.207} C_VEL
LIN {X 0,Y 736.054,Z 389.537,A -85,B 0,C 180,E1 33813.363,E2 33813.363} C_VEL
LIN {X 0,Y 736.093,Z 389.536,A -85,B 0,C 180,E1 33810.543,E2 33810.543} C_VEL
LIN {X 0,Y 736.067,Z 389.535,A -85,B 0,C 180,E1 33807.641,E2 33807.641} C_VEL
LIN {X 0,Y 736.062,Z 389.54,A -85,B 0,C 180,E1 33804.832,E2 33804.832} C_VEL
LIN {X 0,Y 736.098,Z 389.535,A -85,B 0,C 180,E1 33801.825,E2 33801.825} C_VEL
LIN {X 0,Y 736.048,Z 389.541,A -85,B 0,C 180,E1 33798.994,E2 33798.994} C_VEL
LIN {X 0,Y 736.088,Z 389.545,A -85,B 0,C 180,E1 33796.257,E2 33796.257} C_VEL
LIN {X 0,Y 736.077,Z 389.683,A -85,B 0,C 180,E1 33795.12,E2 33795.12} C_VEL
LIN {X 0,Y 737.203,Z 392.799,A -85,B 0,C 180,E1 33794.817,E2 33794.817} C_VEL
LIN {X 0,Y 740.41,Z 399.692,A -85,B 0,C 180,E1 33794.102,E2 33794.102} C_VEL
LIN {X 0,Y 740.25,Z 428.168,A -85,B 0,C 180,E1 33792.243,E2 33792.243} C_VEL
LIN {X 0,Y 741.809,Z 434.836,A -85,B 0,C 180,E1 33792.049,E2 33792.049} C_VEL
LIN {X 0,Y 741.127,Z 649.61,A -85,B 0,C 180,E1 33789.405,E2 33789.405} C_VEL
LIN {X 0,Y 740.468,Z 875.577,A -85,B 0,C 180,E1 33786.719,E2 33786.719} C_VEL
LIN {X 0,Y 740.314,Z 911.677,A -85,B 0,C 180,E1 33786.258,E2 33786.258} C_VEL
LIN {X 0,Y 740.066,Z 938.531,A -85,B 0,C 180,E1 33785.756,E2 33785.756} C_VEL
LIN {X 0,Y 739.794,Z 964.502,A -85,B 0,C 180,E1 33785.118,E2 33785.118} C_VEL
LIN {X 0,Y 739.445,Z 993.127,A -85,B 0,C 180,E1 33784.232,E2 33784.232} C_VEL
LIN {X 0,Y 739.093,Z 1016.411,A -85,B 0,C 180,E1 33783.365,E2 33783.365} C_VEL
LIN {X 0,Y 738.791,Z 1037.626,A -85,B 0,C 180,E1 33782.456,E2 33782.456} C_VEL
LIN {X 0,Y 738.487,Z 1058.254,A -85,B 0,C 180,E1 33781.46,E2 33781.46} C_VEL
LIN {X 0,Y 738.112,Z 1082.643,A -85,B 0,C 180,E1 33780.128,E2 33780.128} C_VEL
LIN {X 0,Y 737.733,Z 1103.861,A -85,B 0,C 180,E1 33778.807,E2 33778.807} C_VEL
LIN {X 0,Y 737.462,Z 1122.302,A -85,B 0,C 180,E1 33777.535,E2 33777.535} C_VEL
LIN {X 0,Y 737.182,Z 1143.229,A -85,B 0,C 180,E1 33775.937,E2 33775.937} C_VEL
LIN {X 0,Y 736.844,Z 1162.156,A -85,B 0,C 180,E1 33774.304,E2 33774.304} C_VEL
LIN {X 0,Y 736.681,Z 1177.566,A -85,B 0,C 180,E1 33772.838,E2 33772.838} C_VEL
LIN {X 0,Y 736.483,Z 1194.962,A -85,B 0,C 180,E1 33771.006,E2 33771.006} C_VEL
LIN {X 0,Y 736.294,Z 1210.133,A -85,B 0,C 180,E1 33769.189,E2 33769.189} C_VEL
LIN {X 0,Y 736.156,Z 1221.812,A -85,B 0,C 180,E1 33767.634,E2 33767.634} C_VEL
LIN {X 0,Y 736.081,Z 1232.24,A -85,B 0,C 180,E1 33766.091,E2 33766.091} C_VEL
LIN {X 0,Y 736.047,Z 1242.438,A -85,B 0,C 180,E1 33764.397,E2 33764.397} C_VEL
LIN {X 0,Y 735.956,Z 1253.985,A -85,B 0,C 180,E1 33762.16,E2 33762.16} C_VEL
LIN {X 0,Y 735.948,Z 1261.808,A -85,B 0,C 180,E1 33760.334,E2 33760.334} C_VEL
LIN {X 0,Y 735.92,Z 1267.781,A -85,B 0,C 180,E1 33758.677,E2 33758.677} C_VEL
LIN {X 0,Y 735.913,Z 1273.167,A -85,B 0,C 180,E1 33756.87,E2 33756.87} C_VEL
LIN {X 0,Y 735.909,Z 1277.776,A -85,B 0,C 180,E1 33754.758,E2 33754.758} C_VEL
LIN {X 0,Y 735.915,Z 1280.47,A -85,B 0,C 180,E1 33752.807,E2 33752.807} C_VEL
LIN {X 0,Y 735.874,Z 1281.714,A -85,B 0,C 180,E1 33751.016,E2 33751.016} C_VEL
LIN {X 0,Y 735.863,Z 1281.828,A -85,B 0,C 180,E1 33749.381,E2 33749.381} C_VEL
LIN {X 0,Y 735.908,Z 1280.949,A -85,B 0,C 180,E1 33747.745,E2 33747.745} C_VEL
LIN {X 0,Y 735.918,Z 1278.809,A -85,B 0,C 180,E1 33745.874,E2 33745.874} C_VEL
LIN {X 0,Y 735.923,Z 1274.743,A -85,B 0,C 180,E1 33743.764,E2 33743.764} C_VEL
LIN {X 0,Y 735.931,Z 1269.085,A -85,B 0,C 180,E1 33741.724,E2 33741.724} C_VEL
LIN {X 0,Y 735.945,Z 1263.06,A -85,B 0,C 180,E1 33739.989,E2 33739.989} C_VEL
LIN {X 0,Y 735.951,Z 1256.162,A -85,B 0,C 180,E1 33738.325,E2 33738.325} C_VEL
LIN {X 0,Y 735.966,Z 1248.904,A -85,B 0,C 180,E1 33736.811,E2 33736.811} C_VEL
LIN {X 0,Y 736.041,Z 1240.154,A -85,B 0,C 180,E1 33735.208,E2 33735.208} C_VEL
LIN {X 0,Y 736.1,Z 1230.198,A -85,B 0,C 180,E1 33733.593,E2 33733.593} C_VEL
LIN {X 0,Y 736.256,Z 1216.616,A -85,B 0,C 180,E1 33731.64,E2 33731.64} C_VEL
LIN {X 0,Y 736.373,Z 1201.422,A -85,B 0,C 180,E1 33729.747,E2 33729.747} C_VEL
LIN {X 0,Y 736.537,Z 1187.744,A -85,B 0,C 180,E1 33728.213,E2 33728.213} C_VEL
LIN {X 0,Y 736.753,Z 1171.417,A -85,B 0,C 180,E1 33726.555,E2 33726.555} C_VEL
LIN {X 0,Y 737.034,Z 1151.892,A -85,B 0,C 180,E1 33724.793,E2 33724.793} C_VEL
LIN {X 0,Y 737.238,Z 1135.012,A -85,B 0,C 180,E1 33723.418,E2 33723.418} C_VEL
LIN {X 0,Y 737.58,Z 1115.673,A -85,B 0,C 180,E1 33721.989,E2 33721.989} C_VEL
LIN {X 0,Y 737.953,Z 1092.087,A -85,B 0,C 180,E1 33720.445,E2 33720.445} C_VEL
LIN {X 0,Y 738.232,Z 1072.521,A -85,B 0,C 180,E1 33719.301,E2 33719.301} C_VEL
LIN {X 0,Y 738.551,Z 1052.071,A -85,B 0,C 180,E1 33718.227,E2 33718.227} C_VEL
LIN {X 0,Y 739.014,Z 1026.679,A -85,B 0,C 180,E1 33717.056,E2 33717.056} C_VEL
LIN {X 0,Y 739.316,Z 1003.478,A -85,B 0,C 180,E1 33716.141,E2 33716.141} C_VEL
LIN {X 0,Y 739.58,Z 982.463,A -85,B 0,C 180,E1 33715.422,E2 33715.422} C_VEL
LIN {X 0,Y 739.856,Z 959.788,A -85,B 0,C 180,E1 33714.756,E2 33714.756} C_VEL
LIN {X 0,Y 740.129,Z 932.848,A -85,B 0,C 180,E1 33714.124,E2 33714.124} C_VEL
